LIN {X 0,Y 523.952,Z 221.716,A -85,B 0,C 180,E1 -4742.867,E2 -4742.867} C_VEL
LIN {X 0,Y 523.943,Z 221.723,A -85,B 0,C 180,E1 -4745.803,E2 -4745.803} C_VEL
LIN {X 0,Y 523.98,Z 221.883,A -85,B 0,C 180,E1 -4746.587,E2 -4746.587} C_VEL
LIN {X 0,Y 525.207,Z 229.637,A -85,B 0,C 180,E1 -4747.995,E2 -4747.995} C_VEL
LIN {X 0,Y 524.785,Z 247.797,A -85,B 0,C 180,E1 -4751.048,E2 -4751.048} C_VEL
LIN {X 0,Y 524.373,Z 265.937,A -85,B 0,C 180,E1 -4754.052,E2 -4754.052} C_VEL
LIN {X 0,Y 524.299,Z 270.906,A -85,B 0,C 180,E1 -4754.827,E2 -4754.827} C_VEL
LIN {X 0,Y 525.932,Z 281.44,A -85,B 0,C 180,E1 -4755.046,E2 -4755.046} C_VEL
LIN {X 0,Y 525.541,Z 378.256,A -85,B 0,C 180,E1 -4756.391,E2 -4756.391} C_VEL
LIN {X 0,Y 525.328,Z 391.632,A -85,B 0,C 180,E1 -4756.731,E2 -4756.731} C_VEL
LIN {X 0,Y 525.042,Z 404.968,A -85,B 0,C 180,E1 -4757.24,E2 -4757.24} C_VEL
LIN {X 0,Y 524.817,Z 416.488,A -85,B 0,C 180,E1 -4757.844,E2 -4757.844} C_VEL
LIN {X 0,Y 524.548,Z 427.759,A -85,B 0,C 180,E1 -4758.601,E2 -4758.601} C_VEL
LIN {X 0,Y 524.211,Z 438.203,A -85,B 0,C 180,E1 -4759.474,E2 -4759.474} C_VEL
LIN {X 0,Y 524.027,Z 446.741,A -85,B 0,C 180,E1 -4760.349,E2 -4760.349} C_VEL
LIN {X 0,Y 523.818,Z 454.616,A -85,B 0,C 180,E1 -4761.318,E2 -4761.318} C_VEL
LIN {X 0,Y 523.623,Z 462.304,A -85,B 0,C 180,E1 -4762.48,E2 -4762.48} C_VEL
LIN {X 0,Y 523.495,Z 469.387,A -85,B 0,C 180,E1 -4763.834,E2 -4763.834} C_VEL
LIN {X 0,Y 523.384,Z 474.097,A -85,B 0,C 180,E1 -4764.992,E2 -4764.992} C_VEL
LIN {X 0,Y 523.444,Z 477.697,A -85,B 0,C 180,E1 -4766.15,E2 -4766.15} C_VEL
LIN {X 0,Y 523.369,Z 479.553,A -85,B 0,C 180,E1 -4766.92,E2 -4766.92} C_VEL
LIN {X 0,Y 523.335,Z 480.944,A -85,B 0,C 180,E1 -4767.69,E2 -4767.69} C_VEL
LIN {X 0,Y 523.25,Z 482.542,A -85,B 0,C 180,E1 -4769.23,E2 -4769.23} C_VEL
LIN {X 0,Y 523.247,Z 482.758,A -85,B 0,C 180,E1 -4769.999,E2 -4769.999} C_VEL
LIN {X 0,Y 523.275,Z 481.938,A -85,B 0,C 180,E1 -4771.539,E2 -4771.539} C_VEL
LIN {X 0,Y 523.335,Z 480.947,A -85,B 0,C 180,E1 -4772.308,E2 -4772.308} C_VEL
LIN {X 0,Y 523.368,Z 479.556,A -85,B 0,C 180,E1 -4773.078,E2 -4773.078} C_VEL
LIN {X 0,Y 523.424,Z 476.63,A -85,B 0,C 180,E1 -4774.234,E2 -4774.234} C_VEL
LIN {X 0,Y 523.462,Z 472.667,A -85,B 0,C 180,E1 -4775.392,E2 -4775.392} C_VEL
LIN {X 0,Y 523.504,Z 466.596,A -85,B 0,C 180,E1 -4776.74,E2 -4776.74} C_VEL
LIN {X 0,Y 523.674,Z 459.907,A -85,B 0,C 180,E1 -4777.906,E2 -4777.906} C_VEL
LIN {X 0,Y 523.861,Z 451.635,A -85,B 0,C 180,E1 -4779.069,E2 -4779.069} C_VEL
LIN {X 0,Y 524.081,Z 443.153,A -85,B 0,C 180,E1 -4780.039,E2 -4780.039} C_VEL
LIN {X 0,Y 524.369,Z 432.668,A -85,B 0,C 180,E1 -4781.01,E2 -4781.01} C_VEL
LIN {X 0,Y 524.657,Z 422.414,A -85,B 0,C 180,E1 -4781.778,E2 -4781.778} C_VEL
LIN {X 0,Y 524.934,Z 410.912,A -85,B 0,C 180,E1 -4782.467,E2 -4782.467} C_VEL
LIN {X 0,Y 525.17,Z 399.214,A -85,B 0,C 180,E1 -4783.002,E2 -4783.002} C_VEL
LIN {X 0,Y 525.408,Z 386.643,A -85,B 0,C 180,E1 -4783.414,E2 -4783.414} C_VEL
LIN {X 0,Y 525.557,Z 373.865,A -85,B 0,C 180,E1 -4783.681,E2 -4783.681} C_VEL
LIN {X 0,Y 525.798,Z 280.337,A -85,B 0,C 180,E1 -4784.973,E2 -4784.973} C_VEL
LIN {X 0,Y 524.296,Z 270.856,A -85,B 0,C 180,E1 -4785.172,E2 -4785.172} C_VEL
LIN {X 0,Y 524.447,Z 259.751,A -85,B 0,C 180,E1 -4786.945,E2 -4786.945} C_VEL
LIN {X 0,Y 524.832,Z 242.691,A -85,B 0,C 180,E1 -4789.762,E2 -4789.762} C_VEL
LIN {X 0,Y 525.171,Z 229.26,A -85,B 0,C 180,E1 -4792.005,E2 -4792.005} C_VEL
LIN {X 0,Y 523.968,Z 221.828,A -85,B 0,C 180,E1 -4793.36,E2 -4793.36} C_VEL
LIN {X 0,Y 523.945,Z 221.72,A -85,B 0,C 180,E1 -4796.272,E2 -4796.272} C_VEL
LIN {X 0,Y 523.932,Z 221.718,A -85,B 0,C 180,E1 -4798.874,E2 -4798.874} C_VEL
LIN {X 0,Y 523.922,Z 221.723,A -85,B 0,C 180,E1 -4801.543,E2 -4801.543} C_VEL
LIN {X 0,Y 523.934,Z 221.722,A -85,B 0,C 180,E1 -4804.289,E2 -4804.289} C_VEL
LIN {X 0,Y 523.906,Z 221.718,A -85,B 0,C 180,E1 -4807.131,E2 -4807.131} C_VEL
LIN {X 0,Y 523.914,Z 221.724,A -85,B 0,C 180,E1 -4810.125,E2 -4810.125} C_VEL
LIN {X 0,Y 523.917,Z 221.723,A -85,B 0,C 180,E1 -4812.455,E2 -4812.455} C_VEL
LIN {X 0,Y 523.938,Z 221.715,A -85,B 0,C 180,E1 -4815.309,E2 -4815.309} C_VEL
LIN {X 0,Y 523.941,Z 221.72,A -85,B 0,C 180,E1 -4818.69,E2 -4818.69} C_VEL
LIN {X 0,Y 523.912,Z 221.719,A -85,B 0,C 180,E1 -4821.896,E2 -4821.896} C_VEL
LIN {X 0,Y 523.918,Z 221.722,A -85,B 0,C 180,E1 -4824.91,E2 -4824.91} C_VEL
LIN {X 0,Y 523.933,Z 221.716,A -85,B 0,C 180,E1 -4827.678,E2 -4827.678} C_VEL
LIN {X 0,Y 523.934,Z 221.725,A -85,B 0,C 180,E1 -4830.678,E2 -4830.678} C_VEL
LIN {X 0,Y 523.9,Z 221.72,A -85,B 0,C 180,E1 -4833.723,E2 -4833.723} C_VEL
LIN {X 0,Y 523.905,Z 221.72,A -85,B 0,C 180,E1 -4836.267,E2 -4836.267} C_VEL
LIN {X 0,Y 523.939,Z 221.721,A -85,B 0,C 180,E1 -4838.764,E2 -4838.764} C_VEL
LIN {X 0,Y 523.927,Z 221.721,A -85,B 0,C 180,E1 -4841.218,E2 -4841.218} C_VEL
LIN {X 0,Y 523.903,Z 221.722,A -85,B 0,C 180,E1 -4843.636,E2 -4843.636} C_VEL
LIN {X 0,Y 523.906,Z 221.717,A -85,B 0,C 180,E1 -4846.025,E2 -4846.025} C_VEL
LIN {X 0,Y 524.008,Z 221.706,A -85,B 0,C 180,E1 -4848.392,E2 -4848.392} C_VEL
LIN {X 0,Y 523.938,Z 221.721,A -85,B 0,C 180,E1 -4851.513,E2 -4851.513} C_VEL
LIN {X 0,Y 524.002,Z 221.711,A -85,B 0,C 180,E1 -4853.838,E2 -4853.838} C_VEL
LIN {X 0,Y 523.937,Z 221.723,A -85,B 0,C 180,E1 -4855.381,E2 -4855.381} C_VEL
LIN {X 0,Y 524.087,Z 221.704,A -85,B 0,C 180,E1 -4857.692,E2 -4857.692} C_VEL
LIN {X 0,Y 524.076,Z 221.7,A -85,B 0,C 180,E1 -4859.997,E2 -4859.997} C_VEL
LIN {X 0,Y 524.083,Z 221.698,A -85,B 0,C 180,E1 -4862.303,E2 -4862.303} C_VEL
LIN {X 0,Y 523.981,Z 221.713,A -85,B 0,C 180,E1 -4866.157,E2 -4866.157} C_VEL
LIN {X 0,Y 523.93,Z 221.718,A -85,B 0,C 180,E1 -4869.26,E2 -4869.26} C_VEL
LIN {X 0,Y 523.931,Z 221.719,A -85,B 0,C 180,E1 -4872.39,E2 -4872.39} C_VEL
LIN {X 0,Y 523.911,Z 221.723,A -85,B 0,C 180,E1 -4875.559,E2 -4875.559} C_VEL
LIN {X 0,Y 523.897,Z 221.727,A -85,B 0,C 180,E1 -4877.968,E2 -4877.968} C_VEL
LIN {X 0,Y 523.952,Z 221.719,A -85,B 0,C 180,E1 -4880.407,E2 -4880.407} C_VEL
LIN {X 0,Y 523.889,Z 221.722,A -85,B 0,C 180,E1 -4882.891,E2 -4882.891} C_VEL
LIN {X 0,Y 523.906,Z 221.719,A -85,B 0,C 180,E1 -4885.417,E2 -4885.417} C_VEL
LIN {X 0,Y 523.901,Z 221.725,A -85,B 0,C 180,E1 -4887.999,E2 -4887.999} C_VEL
LIN {X 0,Y 523.914,Z 221.722,A -85,B 0,C 180,E1 -4890.851,E2 -4890.851} C_VEL
LIN {X 0,Y 523.935,Z 221.717,A -85,B 0,C 180,E1 -4893.732,E2 -4893.732} C_VEL
LIN {X 0,Y 523.894,Z 221.728,A -85,B 0,C 180,E1 -4896.402,E2 -4896.402} C_VEL
LIN {X 0,Y 523.903,Z 221.725,A -85,B 0,C 180,E1 -4899.081,E2 -4899.081} C_VEL
LIN {X 0,Y 523.943,Z 221.719,A -85,B 0,C 180,E1 -4901.31,E2 -4901.31} C_VEL
LIN {X 0,Y 523.93,Z 221.726,A -85,B 0,C 180,E1 -4904.69,E2 -4904.69} C_VEL
LIN {X 0,Y 524.01,Z 221.942,A -85,B 0,C 180,E1 -4905.694,E2 -4905.694} C_VEL
LIN {X 0,Y 523.765,Z 225.215,A -85,B 0,C 180,E1 -4906.283,E2 -4906.283} C_VEL
LIN {X 0,Y 522.413,Z 228.497,A -85,B 0,C 180,E1 -4906.811,E2 -4906.811} C_VEL
LIN {X 0,Y 518.311,Z 236.117,A -85,B 0,C 180,E1 -4907.987,E2 -4907.987} C_VEL
LIN {X 0,Y 517.523,Z 239.242,A -85,B 0,C 180,E1 -4908.526,E2 -4908.526} C_VEL
LIN {X 0,Y 517.224,Z 256.986,A -85,B 0,C 180,E1 -4911.626,E2 -4911.626} C_VEL
LIN {X 0,Y 517.434,Z 258.712,A -85,B 0,C 180,E1 -4911.713,E2 -4911.713} C_VEL
LIN {X 0,Y 519.065,Z 267.751,A -85,B 0,C 180,E1 -4911.893,E2 -4911.893} C_VEL
LIN {X 0,Y 518.601,Z 364.846,A -85,B 0,C 180,E1 -4913.266,E2 -4913.266} C_VEL
LIN {X 0,Y 518.415,Z 377.895,A -85,B 0,C 180,E1 -4913.608,E2 -4913.608} C_VEL
LIN {X 0,Y 518.212,Z 390.252,A -85,B 0,C 180,E1 -4914.088,E2 -4914.088} C_VEL
LIN {X 0,Y 517.944,Z 401.526,A -85,B 0,C 180,E1 -4914.675,E2 -4914.675} C_VEL
LIN {X 0,Y 517.559,Z 412.829,A -85,B 0,C 180,E1 -4915.432,E2 -4915.432} C_VEL
LIN {X 0,Y 517.306,Z 422.833,A -85,B 0,C 180,E1 -4916.268,E2 -4916.268} C_VEL
LIN {X 0,Y 516.997,Z 432.757,A -85,B 0,C 180,E1 -4917.288,E2 -4917.288} C_VEL
LIN {X 0,Y 516.75,Z 441.634,A -85,B 0,C 180,E1 -4918.426,E2 -4918.426} C_VEL
LIN {X 0,Y 516.58,Z 448.883,A -85,B 0,C 180,E1 -4919.575,E2 -4919.575} C_VEL
LIN {X 0,Y 516.438,Z 454.473,A -85,B 0,C 180,E1 -4920.666,E2 -4920.666} C_VEL
LIN {X 0,Y 516.346,Z 459.559,A -85,B 0,C 180,E1 -4921.917,E2 -4921.917} C_VEL
LIN {X 0,Y 516.277,Z 463.773,A -85,B 0,C 180,E1 -4923.307,E2 -4923.307} C_VEL
LIN {X 0,Y 516.231,Z 465.648,A -85,B 0,C 180,E1 -4924.174,E2 -4924.174} C_VEL
LIN {X 0,Y 516.18,Z 467.035,A -85,B 0,C 180,E1 -4925.035,E2 -4925.035} C_VEL
LIN {X 0,Y 516.196,Z 467.919,A -85,B 0,C 180,E1 -4925.893,E2 -4925.893} C_VEL
LIN {X 0,Y 516.165,Z 468.305,A -85,B 0,C 180,E1 -4926.744,E2 -4926.744} C_VEL
LIN {X 0,Y 516.156,Z 468.166,A -85,B 0,C 180,E1 -4927.791,E2 -4927.791} C_VEL
LIN {X 0,Y 516.192,Z 466.722,A -85,B 0,C 180,E1 -4929.269,E2 -4929.269} C_VEL
LIN {X 0,Y 516.243,Z 465.293,A -85,B 0,C 180,E1 -4930.103,E2 -4930.103} C_VEL
LIN {X 0,Y 516.303,Z 462.244,A -85,B 0,C 180,E1 -4931.345,E2 -4931.345} C_VEL
LIN {X 0,Y 516.37,Z 458.075,A -85,B 0,C 180,E1 -4932.578,E2 -4932.578} C_VEL
LIN {X 0,Y 516.489,Z 451.624,A -85,B 0,C 180,E1 -4934.006,E2 -4934.006} C_VEL
LIN {X 0,Y 516.676,Z 444.589,A -85,B 0,C 180,E1 -4935.225,E2 -4935.225} C_VEL
LIN {X 0,Y 516.902,Z 437.397,A -85,B 0,C 180,E1 -4936.236,E2 -4936.236} C_VEL
LIN {X 0,Y 517.134,Z 428.727,A -85,B 0,C 180,E1 -4937.242,E2 -4937.242} C_VEL
LIN {X 0,Y 517.418,Z 418.012,A -85,B 0,C 180,E1 -4938.245,E2 -4938.245} C_VEL
LIN {X 0,Y 517.736,Z 407.363,A -85,B 0,C 180,E1 -4939.045,E2 -4939.045} C_VEL
LIN {X 0,Y 518.067,Z 395.552,A -85,B 0,C 180,E1 -4939.744,E2 -4939.744} C_VEL
LIN {X 0,Y 518.294,Z 383.305,A -85,B 0,C 180,E1 -4940.291,E2 -4940.291} C_VEL
LIN {X 0,Y 518.591,Z 370.453,A -85,B 0,C 180,E1 -4940.696,E2 -4940.696} C_VEL
LIN {X 0,Y 518.685,Z 357.828,A -85,B 0,C 180,E1 -4940.941,E2 -4940.941} C_VEL
LIN {X 0,Y 519.021,Z 267.402,A -85,B 0,C 180,E1 -4942.203,E2 -4942.203} C_VEL
LIN {X 0,Y 517.278,Z 257.789,A -85,B 0,C 180,E1 -4942.409,E2 -4942.409} C_VEL
LIN {X 0,Y 517.234,Z 256.652,A -85,B 0,C 180,E1 -4942.539,E2 -4942.539} C_VEL
LIN {X 0,Y 517.566,Z 244.544,A -85,B 0,C 180,E1 -4944.742,E2 -4944.742} C_VEL
LIN {X 0,Y 517.918,Z 228.732,A -85,B 0,C 180,E1 -4947.668,E2 -4947.668} C_VEL
LIN {X 0,Y 516.991,Z 222.635,A -85,B 0,C 180,E1 -4948.905,E2 -4948.905} C_VEL
LIN {X 0,Y 517.058,Z 222.578,A -85,B 0,C 180,E1 -4950.779,E2 -4950.779} C_VEL
LIN {X 0,Y 516.981,Z 222.589,A -85,B 0,C 180,E1 -4953.118,E2 -4953.118} C_VEL
LIN {X 0,Y 516.966,Z 222.585,A -85,B 0,C 180,E1 -4956.244,E2 -4956.244} C_VEL
LIN {X 0,Y 516.915,Z 222.597,A -85,B 0,C 180,E1 -4959.391,E2 -4959.391} C_VEL
LIN {X 0,Y 516.946,Z 222.591,A -85,B 0,C 180,E1 -4961.826,E2 -4961.826} C_VEL
LIN {X 0,Y 516.906,Z 222.593,A -85,B 0,C 180,E1 -4965.147,E2 -4965.147} C_VEL
LIN {X 0,Y 516.889,Z 222.598,A -85,B 0,C 180,E1 -4968.224,E2 -4968.224} C_VEL
LIN {X 0,Y 516.876,Z 222.595,A -85,B 0,C 180,E1 -4970.703,E2 -4970.703} C_VEL
LIN {X 0,Y 516.856,Z 222.604,A -85,B 0,C 180,E1 -4974.075,E2 -4974.075} C_VEL
LIN {X 0,Y 516.863,Z 222.599,A -85,B 0,C 180,E1 -4976.662,E2 -4976.662} C_VEL
LIN {X 0,Y 516.878,Z 222.591,A -85,B 0,C 180,E1 -4979.526,E2 -4979.526} C_VEL
LIN {X 0,Y 516.863,Z 222.602,A -85,B 0,C 180,E1 -4982.546,E2 -4982.546} C_VEL
LIN {X 0,Y 516.826,Z 222.596,A -85,B 0,C 180,E1 -4985.331,E2 -4985.331} C_VEL
LIN {X 0,Y 516.844,Z 222.606,A -85,B 0,C 180,E1 -4988.72,E2 -4988.72} C_VEL
LIN {X 0,Y 516.826,Z 222.598,A -85,B 0,C 180,E1 -4991.784,E2 -4991.784} C_VEL
LIN {X 0,Y 516.871,Z 222.601,A -85,B 0,C 180,E1 -4995.01,E2 -4995.01} C_VEL
LIN {X 0,Y 516.832,Z 222.603,A -85,B 0,C 180,E1 -4998.409,E2 -4998.409} C_VEL
LIN {X 0,Y 516.855,Z 222.595,A -85,B 0,C 180,E1 -5001.287,E2 -5001.287} C_VEL
LIN {X 0,Y 516.85,Z 222.597,A -85,B 0,C 180,E1 -5004.223,E2 -5004.223} C_VEL
LIN {X 0,Y 516.863,Z 222.605,A -85,B 0,C 180,E1 -5007.055,E2 -5007.055} C_VEL
LIN {X 0,Y 516.838,Z 222.595,A -85,B 0,C 180,E1 -5009.797,E2 -5009.797} C_VEL
LIN {X 0,Y 516.855,Z 222.59,A -85,B 0,C 180,E1 -5012.467,E2 -5012.467} C_VEL
LIN {X 0,Y 516.859,Z 222.603,A -85,B 0,C 180,E1 -5015.649,E2 -5015.649} C_VEL
LIN {X 0,Y 516.875,Z 222.594,A -85,B 0,C 180,E1 -5018.465,E2 -5018.465} C_VEL
LIN {X 0,Y 516.881,Z 222.59,A -85,B 0,C 180,E1 -5020.958,E2 -5020.958} C_VEL
LIN {X 0,Y 516.875,Z 222.589,A -85,B 0,C 180,E1 -5023.412,E2 -5023.412} C_VEL
LIN {X 0,Y 516.876,Z 222.602,A -85,B 0,C 180,E1 -5025.836,E2 -5025.836} C_VEL
LIN {X 0,Y 516.922,Z 222.592,A -85,B 0,C 180,E1 -5028.236,E2 -5028.236} C_VEL
LIN {X 0,Y 516.926,Z 222.588,A -85,B 0,C 180,E1 -5031.402,E2 -5031.402} C_VEL
LIN {X 0,Y 516.983,Z 222.575,A -85,B 0,C 180,E1 -5034.542,E2 -5034.542} C_VEL
LIN {X 0,Y 517.071,Z 222.571,A -85,B 0,C 180,E1 -5037.666,E2 -5037.666} C_VEL
LIN {X 0,Y 517.068,Z 222.572,A -85,B 0,C 180,E1 -5040.781,E2 -5040.781} C_VEL
LIN {X 0,Y 516.946,Z 222.581,A -85,B 0,C 180,E1 -5043.12,E2 -5043.12} C_VEL
LIN {X 0,Y 516.986,Z 222.579,A -85,B 0,C 180,E1 -5046.246,E2 -5046.246} C_VEL
LIN {X 0,Y 516.92,Z 222.589,A -85,B 0,C 180,E1 -5049.392,E2 -5049.392} C_VEL
LIN {X 0,Y 516.959,Z 222.585,A -85,B 0,C 180,E1 -5051.809,E2 -5051.809} C_VEL
LIN {X 0,Y 516.943,Z 222.582,A -85,B 0,C 180,E1 -5055.145,E2 -5055.145} C_VEL
LIN {X 0,Y 516.919,Z 222.59,A -85,B 0,C 180,E1 -5058.225,E2 -5058.225} C_VEL
LIN {X 0,Y 516.911,Z 222.598,A -85,B 0,C 180,E1 -5060.704,E2 -5060.704} C_VEL
LIN {X 0,Y 516.893,Z 222.586,A -85,B 0,C 180,E1 -5064.075,E2 -5064.075} C_VEL
LIN {X 0,Y 516.902,Z 222.594,A -85,B 0,C 180,E1 -5066.661,E2 -5066.661} C_VEL
LIN {X 0,Y 516.894,Z 222.594,A -85,B 0,C 180,E1 -5069.52,E2 -5069.52} C_VEL
LIN {X 0,Y 516.902,Z 222.59,A -85,B 0,C 180,E1 -5072.544,E2 -5072.544} C_VEL
LIN {X 0,Y 516.869,Z 222.605,A -85,B 0,C 180,E1 -5075.329,E2 -5075.329} C_VEL
LIN {X 0,Y 516.886,Z 222.594,A -85,B 0,C 180,E1 -5077.943,E2 -5077.943} C_VEL
LIN {X 0,Y 516.873,Z 222.596,A -85,B 0,C 180,E1 -5080.744,E2 -5080.744} C_VEL
LIN {X 0,Y 516.89,Z 222.599,A -85,B 0,C 180,E1 -5083.904,E2 -5083.904} C_VEL
LIN {X 0,Y 516.89,Z 222.595,A -85,B 0,C 180,E1 -5086.108,E2 -5086.108} C_VEL
LIN {X 0,Y 516.862,Z 222.599,A -85,B 0,C 180,E1 -5089.256,E2 -5089.256} C_VEL
LIN {X 0,Y 516.869,Z 222.6,A -85,B 0,C 180,E1 -5092.274,E2 -5092.274} C_VEL
LIN {X 0,Y 516.889,Z 222.595,A -85,B 0,C 180,E1 -5095.175,E2 -5095.175} C_VEL
LIN {X 0,Y 516.882,Z 222.603,A -85,B 0,C 180,E1 -5097.975,E2 -5097.975} C_VEL
LIN {X 0,Y 516.928,Z 222.592,A -85,B 0,C 180,E1 -5100.695,E2 -5100.695} C_VEL
LIN {X 0,Y 516.91,Z 222.595,A -85,B 0,C 180,E1 -5103.814,E2 -5103.814} C_VEL
LIN {X 0,Y 516.94,Z 222.731,A -85,B 0,C 180,E1 -5106.408,E2 -5106.408} C_VEL
LIN {X 0,Y 518.257,Z 230.758,A -85,B 0,C 180,E1 -5107.894,E2 -5107.894} C_VEL
LIN {X 0,Y 517.843,Z 245.281,A -85,B 0,C 180,E1 -5110.372,E2 -5110.372} C_VEL
LIN {X 0,Y 517.469,Z 261.007,A -85,B 0,C 180,E1 -5113.022,E2 -5113.022} C_VEL
LIN {X 0,Y 517.277,Z 270.787,A -85,B 0,C 180,E1 -5114.614,E2 -5114.614} C_VEL
LIN {X 0,Y 519.075,Z 282.522,A -85,B 0,C 180,E1 -5114.861,E2 -5114.861} C_VEL
LIN {X 0,Y 518.665,Z 378.097,A -85,B 0,C 180,E1 -5116.207,E2 -5116.207} C_VEL
LIN {X 0,Y 518.424,Z 391.496,A -85,B 0,C 180,E1 -5116.551,E2 -5116.551} C_VEL
LIN {X 0,Y 518.128,Z 404.842,A -85,B 0,C 180,E1 -5117.067,E2 -5117.067} C_VEL
LIN {X 0,Y 517.878,Z 416.092,A -85,B 0,C 180,E1 -5117.662,E2 -5117.662} C_VEL
LIN {X 0,Y 517.568,Z 427.645,A -85,B 0,C 180,E1 -5118.446,E2 -5118.446} C_VEL
LIN {X 0,Y 517.206,Z 438.092,A -85,B 0,C 180,E1 -5119.33,E2 -5119.33} C_VEL
LIN {X 0,Y 516.98,Z 446.633,A -85,B 0,C 180,E1 -5120.216,E2 -5120.216} C_VEL
LIN {X 0,Y 516.756,Z 454.51,A -85,B 0,C 180,E1 -5121.198,E2 -5121.198} C_VEL
LIN {X 0,Y 516.551,Z 462.2,A -85,B 0,C 180,E1 -5122.376,E2 -5122.376} C_VEL
LIN {X 0,Y 516.405,Z 469.285,A -85,B 0,C 180,E1 -5123.749,E2 -5123.749} C_VEL
LIN {X 0,Y 516.314,Z 473.997,A -85,B 0,C 180,E1 -5124.923,E2 -5124.923} C_VEL
LIN {X 0,Y 516.353,Z 477.598,A -85,B 0,C 180,E1 -5126.097,E2 -5126.097} C_VEL
LIN {X 0,Y 516.284,Z 479.454,A -85,B 0,C 180,E1 -5126.878,E2 -5126.878} C_VEL
LIN {X 0,Y 516.262,Z 480.846,A -85,B 0,C 180,E1 -5127.659,E2 -5127.659} C_VEL
LIN {X 0,Y 516.16,Z 482.444,A -85,B 0,C 180,E1 -5129.219,E2 -5129.219} C_VEL
LIN {X 0,Y 516.155,Z 482.66,A -85,B 0,C 180,E1 -5129.999,E2 -5129.999} C_VEL
LIN {X 0,Y 516.192,Z 481.839,A -85,B 0,C 180,E1 -5131.56,E2 -5131.56} C_VEL
LIN {X 0,Y 516.261,Z 480.847,A -85,B 0,C 180,E1 -5132.34,E2 -5132.34} C_VEL
LIN {X 0,Y 516.283,Z 479.456,A -85,B 0,C 180,E1 -5133.121,E2 -5133.121} C_VEL
LIN {X 0,Y 516.313,Z 476.528,A -85,B 0,C 180,E1 -5134.293,E2 -5134.293} C_VEL
LIN {X 0,Y 516.398,Z 472.564,A -85,B 0,C 180,E1 -5135.466,E2 -5135.466} C_VEL
LIN {X 0,Y 516.423,Z 467.358,A -85,B 0,C 180,E1 -5136.663,E2 -5136.663} C_VEL
LIN {X 0,Y 516.583,Z 461.034,A -85,B 0,C 180,E1 -5137.818,E2 -5137.818} C_VEL
LIN {X 0,Y 516.772,Z 453.014,A -85,B 0,C 180,E1 -5138.997,E2 -5138.997} C_VEL
LIN {X 0,Y 517.026,Z 444.839,A -85,B 0,C 180,E1 -5139.98,E2 -5139.98} C_VEL
LIN {X 0,Y 517.336,Z 434.868,A -85,B 0,C 180,E1 -5140.963,E2 -5140.963} C_VEL
LIN {X 0,Y 517.646,Z 425.024,A -85,B 0,C 180,E1 -5141.75,E2 -5141.75} C_VEL
LIN {X 0,Y 517.914,Z 413.875,A -85,B 0,C 180,E1 -5142.465,E2 -5142.465} C_VEL
LIN {X 0,Y 518.197,Z 401.437,A -85,B 0,C 180,E1 -5143.08,E2 -5143.08} C_VEL
LIN {X 0,Y 518.502,Z 389.187,A -85,B 0,C 180,E1 -5143.521,E2 -5143.521} C_VEL
LIN {X 0,Y 518.639,Z 376.686,A -85,B 0,C 180,E1 -5143.817,E2 -5143.817} C_VEL
LIN {X 0,Y 519.048,Z 281.84,A -85,B 0,C 180,E1 -5145.149,E2 -5145.149} C_VEL
LIN {X 0,Y 517.261,Z 270.774,A -85,B 0,C 180,E1 -5145.381,E2 -5145.381} C_VEL
LIN {X 0,Y 517.493,Z 259.643,A -85,B 0,C 180,E1 -5147.18,E2 -5147.18} C_VEL
LIN {X 0,Y 517.973,Z 240.109,A -85,B 0,C 180,E1 -5150.452,E2 -5150.452} C_VEL
LIN {X 0,Y 518.205,Z 230.362,A -85,B 0,C 180,E1 -5152.107,E2 -5152.107} C_VEL
LIN {X 0,Y 516.931,Z 222.671,A -85,B 0,C 180,E1 -5153.538,E2 -5153.538} C_VEL
LIN {X 0,Y 516.913,Z 222.594,A -85,B 0,C 180,E1 -5156.657,E2 -5156.657} C_VEL
LIN {X 0,Y 516.912,Z 222.598,A -85,B 0,C 180,E1 -5159.522,E2 -5159.522} C_VEL
LIN {X 0,Y 516.899,Z 222.595,A -85,B 0,C 180,E1 -5162.542,E2 -5162.542} C_VEL
LIN {X 0,Y 516.866,Z 222.599,A -85,B 0,C 180,E1 -5165.328,E2 -5165.328} C_VEL
LIN {X 0,Y 516.88,Z 222.601,A -85,B 0,C 180,E1 -5167.941,E2 -5167.941} C_VEL
LIN {X 0,Y 516.865,Z 222.598,A -85,B 0,C 180,E1 -5170.742,E2 -5170.742} C_VEL
LIN {X 0,Y 516.856,Z 222.599,A -85,B 0,C 180,E1 -5172.833,E2 -5172.833} C_VEL
LIN {X 0,Y 516.897,Z 222.593,A -85,B 0,C 180,E1 -5175.005,E2 -5175.005} C_VEL
LIN {X 0,Y 516.904,Z 222.599,A -85,B 0,C 180,E1 -5178.399,E2 -5178.399} C_VEL
LIN {X 0,Y 516.876,Z 222.594,A -85,B 0,C 180,E1 -5181.282,E2 -5181.282} C_VEL
LIN {X 0,Y 516.866,Z 222.601,A -85,B 0,C 180,E1 -5184.217,E2 -5184.217} C_VEL
LIN {X 0,Y 516.88,Z 222.598,A -85,B 0,C 180,E1 -5187.05,E2 -5187.05} C_VEL
LIN {X 0,Y 516.865,Z 222.596,A -85,B 0,C 180,E1 -5189.793,E2 -5189.793} C_VEL
LIN {X 0,Y 516.873,Z 222.6,A -85,B 0,C 180,E1 -5192.462,E2 -5192.462} C_VEL
LIN {X 0,Y 516.844,Z 222.605,A -85,B 0,C 180,E1 -5195.066,E2 -5195.066} C_VEL
LIN {X 0,Y 516.867,Z 222.596,A -85,B 0,C 180,E1 -5197.619,E2 -5197.619} C_VEL
LIN {X 0,Y 516.916,Z 222.59,A -85,B 0,C 180,E1 -5200.127,E2 -5200.127} C_VEL
LIN {X 0,Y 516.889,Z 222.593,A -85,B 0,C 180,E1 -5202.593,E2 -5202.593} C_VEL
LIN {X 0,Y 516.926,Z 222.597,A -85,B 0,C 180,E1 -5205.027,E2 -5205.027} C_VEL
LIN {X 0,Y 516.961,Z 222.584,A -85,B 0,C 180,E1 -5208.231,E2 -5208.231} C_VEL
LIN {X 0,Y 516.912,Z 222.596,A -85,B 0,C 180,E1 -5211.396,E2 -5211.396} C_VEL
LIN {X 0,Y 516.972,Z 222.587,A -85,B 0,C 180,E1 -5213.754,E2 -5213.754} C_VEL
LIN {X 0,Y 516.931,Z 222.586,A -85,B 0,C 180,E1 -5216.88,E2 -5216.88} C_VEL
LIN {X 0,Y 517.078,Z 222.575,A -85,B 0,C 180,E1 -5219.219,E2 -5219.219} C_VEL
LIN {X 0,Y 517.053,Z 222.574,A -85,B 0,C 180,E1 -5222.334,E2 -5222.334} C_VEL
LIN {X 0,Y 516.962,Z 222.589,A -85,B 0,C 180,E1 -5225.458,E2 -5225.458} C_VEL
LIN {X 0,Y 516.905,Z 222.591,A -85,B 0,C 180,E1 -5228.598,E2 -5228.598} C_VEL
LIN {X 0,Y 516.917,Z 222.598,A -85,B 0,C 180,E1 -5231.793,E2 -5231.793} C_VEL
LIN {X 0,Y 516.922,Z 222.59,A -85,B 0,C 180,E1 -5235.141,E2 -5235.141} C_VEL
LIN {X 0,Y 516.859,Z 222.605,A -85,B 0,C 180,E1 -5238.221,E2 -5238.221} C_VEL
LIN {X 0,Y 516.893,Z 222.595,A -85,B 0,C 180,E1 -5240.699,E2 -5240.699} C_VEL
LIN {X 0,Y 516.868,Z 222.603,A -85,B 0,C 180,E1 -5244.07,E2 -5244.07} C_VEL
LIN {X 0,Y 516.875,Z 222.6,A -85,B 0,C 180,E1 -5246.657,E2 -5246.657} C_VEL
LIN {X 0,Y 516.885,Z 222.593,A -85,B 0,C 180,E1 -5249.521,E2 -5249.521} C_VEL
LIN {X 0,Y 516.87,Z 222.603,A -85,B 0,C 180,E1 -5252.541,E2 -5252.541} C_VEL
LIN {X 0,Y 516.855,Z 222.599,A -85,B 0,C 180,E1 -5255.33,E2 -5255.33} C_VEL
LIN {X 0,Y 516.854,Z 222.599,A -85,B 0,C 180,E1 -5257.941,E2 -5257.941} C_VEL
LIN {X 0,Y 516.875,Z 222.604,A -85,B 0,C 180,E1 -5260.737,E2 -5260.737} C_VEL
LIN {X 0,Y 516.853,Z 222.603,A -85,B 0,C 180,E1 -5263.901,E2 -5263.901} C_VEL
LIN {X 0,Y 516.942,Z 222.726,A -85,B 0,C 180,E1 -5265.535,E2 -5265.535} C_VEL
LIN {X 0,Y 517.7,Z 227.862,A -85,B 0,C 180,E1 -5266.514,E2 -5266.514} C_VEL
LIN {X 0,Y 517.523,Z 239.242,A -85,B 0,C 180,E1 -5268.526,E2 -5268.526} C_VEL
LIN {X 0,Y 516.78,Z 242.514,A -85,B 0,C 180,E1 -5269.073,E2 -5269.073} C_VEL
LIN {X 0,Y 511.465,Z 252.389,A -85,B 0,C 180,E1 -5270.641,E2 -5270.641} C_VEL
LIN {X 0,Y 510.373,Z 255.577,A -85,B 0,C 180,E1 -5271.173,E2 -5271.173} C_VEL
LIN {X 0,Y 510.255,Z 256.657,A -85,B 0,C 180,E1 -5271.35,E2 -5271.35} C_VEL
LIN {X 0,Y 510.286,Z 257.654,A -85,B 0,C 180,E1 -5271.463,E2 -5271.463} C_VEL
LIN {X 0,Y 512.22,Z 268.774,A -85,B 0,C 180,E1 -5271.699,E2 -5271.699} C_VEL
LIN {X 0,Y 511.718,Z 365.201,A -85,B 0,C 180,E1 -5273.084,E2 -5273.084} C_VEL
LIN {X 0,Y 511.501,Z 378.295,A -85,B 0,C 180,E1 -5273.435,E2 -5273.435} C_VEL
LIN {X 0,Y 511.305,Z 390.217,A -85,B 0,C 180,E1 -5273.905,E2 -5273.905} C_VEL
LIN {X 0,Y 510.996,Z 402.179,A -85,B 0,C 180,E1 -5274.54,E2 -5274.54} C_VEL
LIN {X 0,Y 510.601,Z 413.104,A -85,B 0,C 180,E1 -5275.286,E2 -5275.286} C_VEL
LIN {X 0,Y 510.299,Z 423.97,A -85,B 0,C 180,E1 -5276.218,E2 -5276.218} C_VEL
LIN {X 0,Y 509.971,Z 433.267,A -85,B 0,C 180,E1 -5277.201,E2 -5277.201} C_VEL
LIN {X 0,Y 509.697,Z 442.379,A -85,B 0,C 180,E1 -5278.402,E2 -5278.402} C_VEL
LIN {X 0,Y 509.509,Z 449.376,A -85,B 0,C 180,E1 -5279.542,E2 -5279.542} C_VEL
LIN {X 0,Y 509.343,Z 455.299,A -85,B 0,C 180,E1 -5280.738,E2 -5280.738} C_VEL
LIN {X 0,Y 509.254,Z 460.298,A -85,B 0,C 180,E1 -5282.026,E2 -5282.026} C_VEL
LIN {X 0,Y 509.192,Z 464.089,A -85,B 0,C 180,E1 -5283.349,E2 -5283.349} C_VEL
LIN {X 0,Y 509.091,Z 466.647,A -85,B 0,C 180,E1 -5284.663,E2 -5284.663} C_VEL
LIN {X 0,Y 509.096,Z 467.832,A -85,B 0,C 180,E1 -5285.65,E2 -5285.65} C_VEL
LIN {X 0,Y 509.075,Z 468.328,A -85,B 0,C 180,E1 -5286.4,E2 -5286.4} C_VEL
LIN {X 0,Y 509.071,Z 468.34,A -85,B 0,C 180,E1 -5287.652,E2 -5287.652} C_VEL
LIN {X 0,Y 509.075,Z 467.289,A -85,B 0,C 180,E1 -5288.966,E2 -5288.966} C_VEL
LIN {X 0,Y 509.138,Z 465.998,A -85,B 0,C 180,E1 -5289.813,E2 -5289.813} C_VEL
LIN {X 0,Y 509.208,Z 463.223,A -85,B 0,C 180,E1 -5291.075,E2 -5291.075} C_VEL
LIN {X 0,Y 509.265,Z 459.354,A -85,B 0,C 180,E1 -5292.327,E2 -5292.327} C_VEL
LIN {X 0,Y 509.377,Z 454.291,A -85,B 0,C 180,E1 -5293.571,E2 -5293.571} C_VEL
LIN {X 0,Y 509.557,Z 447.491,A -85,B 0,C 180,E1 -5294.881,E2 -5294.881} C_VEL
LIN {X 0,Y 509.799,Z 439.894,A -85,B 0,C 180,E1 -5296.04,E2 -5296.04} C_VEL
LIN {X 0,Y 510.04,Z 431.713,A -85,B 0,C 180,E1 -5297.062,E2 -5297.062} C_VEL
LIN {X 0,Y 510.332,Z 421.743,A -85,B 0,C 180,E1 -5298.079,E2 -5298.079} C_VEL
LIN {X 0,Y 510.645,Z 411.942,A -85,B 0,C 180,E1 -5298.891,E2 -5298.891} C_VEL
LIN {X 0,Y 511.007,Z 401.324,A -85,B 0,C 180,E1 -5299.601,E2 -5299.601} C_VEL
LIN {X 0,Y 511.28,Z 389.722,A -85,B 0,C 180,E1 -5300.207,E2 -5300.207} C_VEL
LIN {X 0,Y 511.539,Z 376.813,A -85,B 0,C 180,E1 -5300.703,E2 -5300.703} C_VEL
LIN {X 0,Y 511.722,Z 364.511,A -85,B 0,C 180,E1 -5301.02,E2 -5301.02} C_VEL
LIN {X 0,Y 512.069,Z 267.751,A -85,B 0,C 180,E1 -5302.41,E2 -5302.41} C_VEL
LIN {X 0,Y 510.277,Z 257.584,A -85,B 0,C 180,E1 -5302.64,E2 -5302.64} C_VEL
LIN {X 0,Y 510.567,Z 246.346,A -85,B 0,C 180,E1 -5304.669,E2 -5304.669} C_VEL
LIN {X 0,Y 510.985,Z 230.504,A -85,B 0,C 180,E1 -5307.636,E2 -5307.636} C_VEL
LIN {X 0,Y 510.001,Z 223.506,A -85,B 0,C 180,E1 -5309.063,E2 -5309.063} C_VEL
LIN {X 0,Y 510.029,Z 223.454,A -85,B 0,C 180,E1 -5310.79,E2 -5310.79} C_VEL
LIN {X 0,Y 509.924,Z 223.468,A -85,B 0,C 180,E1 -5313.161,E2 -5313.161} C_VEL
LIN {X 0,Y 509.917,Z 223.463,A -85,B 0,C 180,E1 -5316.331,E2 -5316.331} C_VEL
LIN {X 0,Y 509.877,Z 223.468,A -85,B 0,C 180,E1 -5318.721,E2 -5318.721} C_VEL
LIN {X 0,Y 509.914,Z 223.465,A -85,B 0,C 180,E1 -5321.932,E2 -5321.932} C_VEL
LIN {X 0,Y 509.857,Z 223.472,A -85,B 0,C 180,E1 -5325.243,E2 -5325.243} C_VEL
LIN {X 0,Y 509.852,Z 223.478,A -85,B 0,C 180,E1 -5328.003,E2 -5328.003} C_VEL
LIN {X 0,Y 509.814,Z 223.474,A -85,B 0,C 180,E1 -5331.004,E2 -5331.004} C_VEL
LIN {X 0,Y 509.787,Z 223.48,A -85,B 0,C 180,E1 -5333.566,E2 -5333.566} C_VEL
LIN {X 0,Y 509.85,Z 223.476,A -85,B 0,C 180,E1 -5336.374,E2 -5336.374} C_VEL
LIN {X 0,Y 509.826,Z 223.472,A -85,B 0,C 180,E1 -5339.754,E2 -5339.754} C_VEL
LIN {X 0,Y 509.815,Z 223.477,A -85,B 0,C 180,E1 -5342.772,E2 -5342.772} C_VEL
LIN {X 0,Y 509.784,Z 223.473,A -85,B 0,C 180,E1 -5345.579,E2 -5345.579} C_VEL
LIN {X 0,Y 509.787,Z 223.485,A -85,B 0,C 180,E1 -5348.344,E2 -5348.344} C_VEL
LIN {X 0,Y 509.781,Z 223.475,A -85,B 0,C 180,E1 -5351.433,E2 -5351.433} C_VEL
LIN {X 0,Y 509.815,Z 223.48,A -85,B 0,C 180,E1 -5354.673,E2 -5354.673} C_VEL
LIN {X 0,Y 509.768,Z 223.481,A -85,B 0,C 180,E1 -5357.509,E2 -5357.509} C_VEL
LIN {X 0,Y 509.811,Z 223.476,A -85,B 0,C 180,E1 -5360.649,E2 -5360.649} C_VEL
LIN {X 0,Y 509.804,Z 223.475,A -85,B 0,C 180,E1 -5363.65,E2 -5363.65} C_VEL
LIN {X 0,Y 509.824,Z 223.475,A -85,B 0,C 180,E1 -5366.541,E2 -5366.541} C_VEL
LIN {X 0,Y 509.808,Z 223.476,A -85,B 0,C 180,E1 -5369.336,E2 -5369.336} C_VEL
LIN {X 0,Y 509.814,Z 223.467,A -85,B 0,C 180,E1 -5372.054,E2 -5372.054} C_VEL
LIN {X 0,Y 509.782,Z 223.477,A -85,B 0,C 180,E1 -5374.703,E2 -5374.703} C_VEL
LIN {X 0,Y 509.815,Z 223.483,A -85,B 0,C 180,E1 -5377.462,E2 -5377.462} C_VEL
LIN {X 0,Y 509.908,Z 223.462,A -85,B 0,C 180,E1 -5379.848,E2 -5379.848} C_VEL
LIN {X 0,Y 509.844,Z 223.461,A -85,B 0,C 180,E1 -5383.177,E2 -5383.177} C_VEL
LIN {X 0,Y 509.847,Z 223.474,A -85,B 0,C 180,E1 -5385.637,E2 -5385.637} C_VEL
LIN {X 0,Y 509.885,Z 223.47,A -85,B 0,C 180,E1 -5388.134,E2 -5388.134} C_VEL
LIN {X 0,Y 509.88,Z 223.465,A -85,B 0,C 180,E1 -5391.282,E2 -5391.282} C_VEL
LIN {X 0,Y 509.92,Z 223.458,A -85,B 0,C 180,E1 -5393.673,E2 -5393.673} C_VEL
LIN {X 0,Y 509.889,Z 223.463,A -85,B 0,C 180,E1 -5396.842,E2 -5396.842} C_VEL
LIN {X 0,Y 509.928,Z 223.465,A -85,B 0,C 180,E1 -5398.423,E2 -5398.423} C_VEL
LIN {X 0,Y 510.02,Z 223.449,A -85,B 0,C 180,E1 -5400.792,E2 -5400.792} C_VEL
LIN {X 0,Y 510.041,Z 223.449,A -85,B 0,C 180,E1 -5402.372,E2 -5402.372} C_VEL
LIN {X 0,Y 509.94,Z 223.457,A -85,B 0,C 180,E1 -5406.333,E2 -5406.333} C_VEL
LIN {X 0,Y 509.882,Z 223.472,A -85,B 0,C 180,E1 -5408.723,E2 -5408.723} C_VEL
LIN {X 0,Y 509.911,Z 223.464,A -85,B 0,C 180,E1 -5411.934,E2 -5411.934} C_VEL
LIN {X 0,Y 509.902,Z 223.458,A -85,B 0,C 180,E1 -5415.244,E2 -5415.244} C_VEL
LIN {X 0,Y 509.864,Z 223.472,A -85,B 0,C 180,E1 -5418.486,E2 -5418.486} C_VEL
LIN {X 0,Y 509.853,Z 223.476,A -85,B 0,C 180,E1 -5421.004,E2 -5421.004} C_VEL
LIN {X 0,Y 509.826,Z 223.467,A -85,B 0,C 180,E1 -5423.566,E2 -5423.566} C_VEL
LIN {X 0,Y 509.883,Z 223.465,A -85,B 0,C 180,E1 -5426.371,E2 -5426.371} C_VEL
LIN {X 0,Y 509.86,Z 223.468,A -85,B 0,C 180,E1 -5429.753,E2 -5429.753} C_VEL
LIN {X 0,Y 509.854,Z 223.47,A -85,B 0,C 180,E1 -5432.77,E2 -5432.77} C_VEL
LIN {X 0,Y 509.829,Z 223.477,A -85,B 0,C 180,E1 -5435.578,E2 -5435.578} C_VEL
LIN {X 0,Y 509.857,Z 223.468,A -85,B 0,C 180,E1 -5438.339,E2 -5438.339} C_VEL
LIN {X 0,Y 509.85,Z 223.479,A -85,B 0,C 180,E1 -5441.428,E2 -5441.428} C_VEL
LIN {X 0,Y 509.849,Z 223.471,A -85,B 0,C 180,E1 -5444.671,E2 -5444.671} C_VEL
LIN {X 0,Y 509.811,Z 223.48,A -85,B 0,C 180,E1 -5447.507,E2 -5447.507} C_VEL
LIN {X 0,Y 509.841,Z 223.472,A -85,B 0,C 180,E1 -5450.647,E2 -5450.647} C_VEL
LIN {X 0,Y 509.818,Z 223.481,A -85,B 0,C 180,E1 -5453.646,E2 -5453.646} C_VEL
LIN {X 0,Y 509.867,Z 223.47,A -85,B 0,C 180,E1 -5456.539,E2 -5456.539} C_VEL
LIN {X 0,Y 509.849,Z 223.471,A -85,B 0,C 180,E1 -5459.334,E2 -5459.334} C_VEL
LIN {X 0,Y 509.892,Z 223.472,A -85,B 0,C 180,E1 -5462.054,E2 -5462.054} C_VEL
LIN {X 0,Y 509.821,Z 223.48,A -85,B 0,C 180,E1 -5464.7,E2 -5464.7} C_VEL
LIN {X 0,Y 509.872,Z 223.582,A -85,B 0,C 180,E1 -5466.223,E2 -5466.223} C_VEL
LIN {X 0,Y 511.287,Z 231.878,A -85,B 0,C 180,E1 -5467.789,E2 -5467.789} C_VEL
LIN {X 0,Y 511.023,Z 242.12,A -85,B 0,C 180,E1 -5469.567,E2 -5469.567} C_VEL
LIN {X 0,Y 510.525,Z 259.705,A -85,B 0,C 180,E1 -5472.577,E2 -5472.577} C_VEL
LIN {X 0,Y 510.281,Z 270.685,A -85,B 0,C 180,E1 -5474.398,E2 -5474.398} C_VEL
LIN {X 0,Y 512.223,Z 283.007,A -85,B 0,C 180,E1 -5474.662,E2 -5474.662} C_VEL
LIN {X 0,Y 511.771,Z 379.1,A -85,B 0,C 180,E1 -5476.043,E2 -5476.043} C_VEL
LIN {X 0,Y 511.497,Z 392.121,A -85,B 0,C 180,E1 -5476.39,E2 -5476.39} C_VEL
LIN {X 0,Y 511.195,Z 404.716,A -85,B 0,C 180,E1 -5476.888,E2 -5476.888} C_VEL
LIN {X 0,Y 510.918,Z 416.09,A -85,B 0,C 180,E1 -5477.498,E2 -5477.498} C_VEL
LIN {X 0,Y 510.602,Z 427.531,A -85,B 0,C 180,E1 -5478.286,E2 -5478.286} C_VEL
LIN {X 0,Y 510.217,Z 437.982,A -85,B 0,C 180,E1 -5479.182,E2 -5479.182} C_VEL
LIN {X 0,Y 509.954,Z 446.525,A -85,B 0,C 180,E1 -5480.08,E2 -5480.08} C_VEL
LIN {X 0,Y 509.69,Z 454.404,A -85,B 0,C 180,E1 -5481.075,E2 -5481.075} C_VEL
LIN {X 0,Y 509.505,Z 462.097,A -85,B 0,C 180,E1 -5482.27,E2 -5482.27} C_VEL
LIN {X 0,Y 509.313,Z 469.183,A -85,B 0,C 180,E1 -5483.661,E2 -5483.661} C_VEL
LIN {X 0,Y 509.248,Z 473.897,A -85,B 0,C 180,E1 -5484.853,E2 -5484.853} C_VEL
LIN {X 0,Y 509.247,Z 477.499,A -85,B 0,C 180,E1 -5486.043,E2 -5486.043} C_VEL
LIN {X 0,Y 509.202,Z 479.356,A -85,B 0,C 180,E1 -5486.835,E2 -5486.835} C_VEL
LIN {X 0,Y 509.162,Z 480.747,A -85,B 0,C 180,E1 -5487.626,E2 -5487.626} C_VEL
LIN {X 0,Y 509.074,Z 482.346,A -85,B 0,C 180,E1 -5489.208,E2 -5489.208} C_VEL
LIN {X 0,Y 509.067,Z 482.561,A -85,B 0,C 180,E1 -5489.999,E2 -5489.999} C_VEL
LIN {X 0,Y 509.113,Z 481.74,A -85,B 0,C 180,E1 -5491.581,E2 -5491.581} C_VEL
LIN {X 0,Y 509.162,Z 480.748,A -85,B 0,C 180,E1 -5492.373,E2 -5492.373} C_VEL
LIN {X 0,Y 509.202,Z 479.356,A -85,B 0,C 180,E1 -5493.164,E2 -5493.164} C_VEL
LIN {X 0,Y 509.206,Z 476.426,A -85,B 0,C 180,E1 -5494.353,E2 -5494.353} C_VEL
LIN {X 0,Y 509.312,Z 472.461,A -85,B 0,C 180,E1 -5495.542,E2 -5495.542} C_VEL
LIN {X 0,Y 509.366,Z 466.461,A -85,B 0,C 180,E1 -5496.914,E2 -5496.914} C_VEL
LIN {X 0,Y 509.561,Z 459.691,A -85,B 0,C 180,E1 -5498.126,E2 -5498.126} C_VEL
LIN {X 0,Y 509.77,Z 451.414,A -85,B 0,C 180,E1 -5499.322,E2 -5499.322} C_VEL
LIN {X 0,Y 510.033,Z 442.925,A -85,B 0,C 180,E1 -5500.319,E2 -5500.319} C_VEL
LIN {X 0,Y 510.4,Z 432.433,A -85,B 0,C 180,E1 -5501.315,E2 -5501.315} C_VEL
LIN {X 0,Y 510.697,Z 421.938,A -85,B 0,C 180,E1 -5502.121,E2 -5502.121} C_VEL
LIN {X 0,Y 511.061,Z 410.657,A -85,B 0,C 180,E1 -5502.811,E2 -5502.811} C_VEL
LIN {X 0,Y 511.337,Z 398.935,A -85,B 0,C 180,E1 -5503.36,E2 -5503.36} C_VEL
LIN {X 0,Y 511.594,Z 386.337,A -85,B 0,C 180,E1 -5503.783,E2 -5503.783} C_VEL
LIN {X 0,Y 511.784,Z 373.5,A -85,B 0,C 180,E1 -5504.056,E2 -5504.056} C_VEL
LIN {X 0,Y 512.172,Z 282.329,A -85,B 0,C 180,E1 -5505.349,E2 -5505.349} C_VEL
LIN {X 0,Y 510.281,Z 270.906,A -85,B 0,C 180,E1 -5505.584,E2 -5505.584} C_VEL
LIN {X 0,Y 510.298,Z 269.126,A -85,B 0,C 180,E1 -5505.808,E2 -5505.808} C_VEL
LIN {X 0,Y 510.718,Z 250.991,A -85,B 0,C 180,E1 -5508.867,E2 -5508.867} C_VEL
LIN {X 0,Y 511.262,Z 232.686,A -85,B 0,C 180,E1 -5511.998,E2 -5511.998} C_VEL
LIN {X 0,Y 510.465,Z 226.531,A -85,B 0,C 180,E1 -5513.108,E2 -5513.108} C_VEL
LIN {X 0,Y 509.887,Z 223.513,A -85,B 0,C 180,E1 -5513.721,E2 -5513.721} C_VEL
LIN {X 0,Y 509.88,Z 223.471,A -85,B 0,C 180,E1 -5517.055,E2 -5517.055} C_VEL
LIN {X 0,Y 509.86,Z 223.477,A -85,B 0,C 180,E1 -5519.75,E2 -5519.75} C_VEL
LIN {X 0,Y 509.876,Z 223.469,A -85,B 0,C 180,E1 -5522.773,E2 -5522.773} C_VEL
LIN {X 0,Y 509.825,Z 223.478,A -85,B 0,C 180,E1 -5525.576,E2 -5525.576} C_VEL
LIN {X 0,Y 509.85,Z 223.476,A -85,B 0,C 180,E1 -5528.337,E2 -5528.337} C_VEL
LIN {X 0,Y 509.845,Z 223.471,A -85,B 0,C 180,E1 -5531.425,E2 -5531.425} C_VEL
LIN {X 0,Y 509.841,Z 223.475,A -85,B 0,C 180,E1 -5534.668,E2 -5534.668} C_VEL
LIN {X 0,Y 509.847,Z 223.477,A -85,B 0,C 180,E1 -5538.103,E2 -5538.103} C_VEL
LIN {X 0,Y 509.833,Z 223.477,A -85,B 0,C 180,E1 -5540.644,E2 -5540.644} C_VEL
LIN {X 0,Y 509.808,Z 223.476,A -85,B 0,C 180,E1 -5543.644,E2 -5543.644} C_VEL
LIN {X 0,Y 509.838,Z 223.48,A -85,B 0,C 180,E1 -5546.536,E2 -5546.536} C_VEL
LIN {X 0,Y 509.832,Z 223.473,A -85,B 0,C 180,E1 -5549.331,E2 -5549.331} C_VEL
LIN {X 0,Y 509.831,Z 223.473,A -85,B 0,C 180,E1 -5552.049,E2 -5552.049} C_VEL
LIN {X 0,Y 509.8,Z 223.483,A -85,B 0,C 180,E1 -5554.698,E2 -5554.698} C_VEL
LIN {X 0,Y 509.822,Z 223.475,A -85,B 0,C 180,E1 -5557.457,E2 -5557.457} C_VEL
LIN {X 0,Y 509.904,Z 223.464,A -85,B 0,C 180,E1 -5559.842,E2 -5559.842} C_VEL
LIN {X 0,Y 509.853,Z 223.479,A -85,B 0,C 180,E1 -5563.171,E2 -5563.171} C_VEL
LIN {X 0,Y 509.838,Z 223.472,A -85,B 0,C 180,E1 -5565.631,E2 -5565.631} C_VEL
LIN {X 0,Y 509.9,Z 223.468,A -85,B 0,C 180,E1 -5568.872,E2 -5568.872} C_VEL
LIN {X 0,Y 509.879,Z 223.466,A -85,B 0,C 180,E1 -5572.075,E2 -5572.075} C_VEL
LIN {X 0,Y 509.954,Z 223.458,A -85,B 0,C 180,E1 -5574.461,E2 -5574.461} C_VEL
LIN {X 0,Y 510.027,Z 223.456,A -85,B 0,C 180,E1 -5577.628,E2 -5577.628} C_VEL
LIN {X 0,Y 510.016,Z 223.451,A -85,B 0,C 180,E1 -5579.997,E2 -5579.997} C_VEL
LIN {X 0,Y 510.023,Z 223.449,A -85,B 0,C 180,E1 -5582.366,E2 -5582.366} C_VEL
LIN {X 0,Y 509.916,Z 223.468,A -85,B 0,C 180,E1 -5585.534,E2 -5585.534} C_VEL
LIN {X 0,Y 509.86,Z 223.476,A -85,B 0,C 180,E1 -5587.92,E2 -5587.92} C_VEL
LIN {X 0,Y 509.847,Z 223.471,A -85,B 0,C 180,E1 -5591.124,E2 -5591.124} C_VEL
LIN {X 0,Y 509.829,Z 223.476,A -85,B 0,C 180,E1 -5593.55,E2 -5593.55} C_VEL
LIN {X 0,Y 509.823,Z 223.483,A -85,B 0,C 180,E1 -5596.001,E2 -5596.001} C_VEL
LIN {X 0,Y 509.819,Z 223.479,A -85,B 0,C 180,E1 -5598.482,E2 -5598.482} C_VEL
LIN {X 0,Y 509.83,Z 223.474,A -85,B 0,C 180,E1 -5600.999,E2 -5600.999} C_VEL
LIN {X 0,Y 509.8,Z 223.477,A -85,B 0,C 180,E1 -5603.561,E2 -5603.561} C_VEL
LIN {X 0,Y 509.861,Z 223.478,A -85,B 0,C 180,E1 -5606.369,E2 -5606.369} C_VEL
LIN {X 0,Y 509.834,Z 223.473,A -85,B 0,C 180,E1 -5609.724,E2 -5609.724} C_VEL
LIN {X 0,Y 509.847,Z 223.477,A -85,B 0,C 180,E1 -5612.771,E2 -5612.771} C_VEL
LIN {X 0,Y 509.815,Z 223.475,A -85,B 0,C 180,E1 -5615.578,E2 -5615.578} C_VEL
LIN {X 0,Y 509.824,Z 223.479,A -85,B 0,C 180,E1 -5618.335,E2 -5618.335} C_VEL
LIN {X 0,Y 509.836,Z 223.476,A -85,B 0,C 180,E1 -5621.422,E2 -5621.422} C_VEL
LIN {X 0,Y 509.826,Z 223.483,A -85,B 0,C 180,E1 -5624.666,E2 -5624.666} C_VEL
LIN {X 0,Y 509.913,Z 223.611,A -85,B 0,C 180,E1 -5625.396,E2 -5625.396} C_VEL
LIN {X 0,Y 510.733,Z 229.532,A -85,B 0,C 180,E1 -5626.527,E2 -5626.527} C_VEL
LIN {X 0,Y 510.49,Z 244.552,A -85,B 0,C 180,E1 -5629.211,E2 -5629.211} C_VEL
LIN {X 0,Y 510.255,Z 256.657,A -85,B 0,C 180,E1 -5631.35,E2 -5631.35} C_VEL
LIN {X 0,Y 509.767,Z 258.344,A -85,B 0,C 180,E1 -5631.456,E2 -5631.456} C_VEL
LIN {X 0,Y 506.544,Z 266.749,A -85,B 0,C 180,E1 -5631.491,E2 -5631.491} C_VEL
LIN {X 0,Y 505.172,Z 272.78,A -85,B 0,C 180,E1 -5631.512,E2 -5631.512} C_VEL
LIN {X 0,Y 504.96,Z 279.207,A -85,B 0,C 180,E1 -5631.592,E2 -5631.592} C_VEL
LIN {X 0,Y 505.274,Z 287.823,A -85,B 0,C 180,E1 -5631.758,E2 -5631.758} C_VEL
LIN {X 0,Y 504.838,Z 365.137,A -85,B 0,C 180,E1 -5632.887,E2 -5632.887} C_VEL
LIN {X 0,Y 504.636,Z 378.174,A -85,B 0,C 180,E1 -5633.239,E2 -5633.239} C_VEL
LIN {X 0,Y 504.367,Z 391.196,A -85,B 0,C 180,E1 -5633.763,E2 -5633.763} C_VEL
LIN {X 0,Y 504.051,Z 402.826,A -85,B 0,C 180,E1 -5634.401,E2 -5634.401} C_VEL
LIN {X 0,Y 503.604,Z 414.238,A -85,B 0,C 180,E1 -5635.204,E2 -5635.204} C_VEL
LIN {X 0,Y 503.281,Z 425.089,A -85,B 0,C 180,E1 -5636.164,E2 -5636.164} C_VEL
LIN {X 0,Y 502.928,Z 434.59,A -85,B 0,C 180,E1 -5637.215,E2 -5637.215} C_VEL
LIN {X 0,Y 502.686,Z 442.329,A -85,B 0,C 180,E1 -5638.26,E2 -5638.26} C_VEL
LIN {X 0,Y 502.444,Z 450.006,A -85,B 0,C 180,E1 -5639.533,E2 -5639.533} C_VEL
LIN {X 0,Y 502.275,Z 455.525,A -85,B 0,C 180,E1 -5640.678,E2 -5640.678} C_VEL
LIN {X 0,Y 502.166,Z 461.056,A -85,B 0,C 180,E1 -5642.166,E2 -5642.166} C_VEL
LIN {X 0,Y 502.098,Z 464.868,A -85,B 0,C 180,E1 -5643.604,E2 -5643.604} C_VEL
LIN {X 0,Y 501.987,Z 467.47,A -85,B 0,C 180,E1 -5645.166,E2 -5645.166} C_VEL
LIN {X 0,Y 501.991,Z 468.226,A -85,B 0,C 180,E1 -5646.047,E2 -5646.047} C_VEL
LIN {X 0,Y 501.975,Z 468.469,A -85,B 0,C 180,E1 -5647.513,E2 -5647.513} C_VEL
LIN {X 0,Y 501.957,Z 467.734,A -85,B 0,C 180,E1 -5648.653,E2 -5648.653} C_VEL
LIN {X 0,Y 502.046,Z 466.386,A -85,B 0,C 180,E1 -5649.691,E2 -5649.691} C_VEL
LIN {X 0,Y 502.129,Z 463.081,A -85,B 0,C 180,E1 -5651.222,E2 -5651.222} C_VEL
LIN {X 0,Y 502.189,Z 459.072,A -85,B 0,C 180,E1 -5652.508,E2 -5652.508} C_VEL
LIN {X 0,Y 502.338,Z 453.984,A -85,B 0,C 180,E1 -5653.752,E2 -5653.752} C_VEL
LIN {X 0,Y 502.526,Z 446.862,A -85,B 0,C 180,E1 -5655.112,E2 -5655.112} C_VEL
LIN {X 0,Y 502.791,Z 439.341,A -85,B 0,C 180,E1 -5656.254,E2 -5656.254} C_VEL
LIN {X 0,Y 503.101,Z 429.85,A -85,B 0,C 180,E1 -5657.424,E2 -5657.424} C_VEL
LIN {X 0,Y 503.415,Z 419.745,A -85,B 0,C 180,E1 -5658.424,E2 -5658.424} C_VEL
LIN {X 0,Y 503.821,Z 407.968,A -85,B 0,C 180,E1 -5659.35,E2 -5659.35} C_VEL
LIN {X 0,Y 504.218,Z 396.286,A -85,B 0,C 180,E1 -5660.068,E2 -5660.068} C_VEL
LIN {X 0,Y 504.493,Z 384.191,A -85,B 0,C 180,E1 -5660.63,E2 -5660.63} C_VEL
LIN {X 0,Y 504.75,Z 371.901,A -85,B 0,C 180,E1 -5661.039,E2 -5661.039} C_VEL
LIN {X 0,Y 504.944,Z 359.104,A -85,B 0,C 180,E1 -5661.307,E2 -5661.307} C_VEL
LIN {X 0,Y 505.235,Z 268.712,A -85,B 0,C 180,E1 -5662.609,E2 -5662.609} C_VEL
LIN {X 0,Y 503.276,Z 257.734,A -85,B 0,C 180,E1 -5662.856,E2 -5662.856} C_VEL
LIN {X 0,Y 503.523,Z 250.288,A -85,B 0,C 180,E1 -5664.193,E2 -5664.193} C_VEL
LIN {X 0,Y 504.035,Z 232.277,A -85,B 0,C 180,E1 -5667.603,E2 -5667.603} C_VEL
LIN {X 0,Y 503.008,Z 224.431,A -85,B 0,C 180,E1 -5669.2,E2 -5669.2} C_VEL
LIN {X 0,Y 502.871,Z 224.347,A -85,B 0,C 180,E1 -5671.602,E2 -5671.602} C_VEL
LIN {X 0,Y 502.867,Z 224.347,A -85,B 0,C 180,E1 -5673.205,E2 -5673.205} C_VEL
LIN {X 0,Y 502.869,Z 224.34,A -85,B 0,C 180,E1 -5676.42,E2 -5676.42} C_VEL
LIN {X 0,Y 502.836,Z 224.346,A -85,B 0,C 180,E1 -5678.845,E2 -5678.845} C_VEL
LIN {X 0,Y 502.856,Z 224.341,A -85,B 0,C 180,E1 -5682.102,E2 -5682.102} C_VEL
LIN {X 0,Y 502.812,Z 224.352,A -85,B 0,C 180,E1 -5685.401,E2 -5685.401} C_VEL
LIN {X 0,Y 502.81,Z 224.353,A -85,B 0,C 180,E1 -5688.124,E2 -5688.124} C_VEL
LIN {X 0,Y 502.794,Z 224.351,A -85,B 0,C 180,E1 -5690.538,E2 -5690.538} C_VEL
LIN {X 0,Y 502.753,Z 224.354,A -85,B 0,C 180,E1 -5693.043,E2 -5693.043} C_VEL
LIN {X 0,Y 502.767,Z 224.355,A -85,B 0,C 180,E1 -5695.68,E2 -5695.68} C_VEL
LIN {X 0,Y 502.764,Z 224.355,A -85,B 0,C 180,E1 -5698.378,E2 -5698.378} C_VEL
LIN {X 0,Y 502.764,Z 224.353,A -85,B 0,C 180,E1 -5701.146,E2 -5701.146} C_VEL
LIN {X 0,Y 502.758,Z 224.357,A -85,B 0,C 180,E1 -5703.998,E2 -5703.998} C_VEL
LIN {X 0,Y 502.722,Z 224.359,A -85,B 0,C 180,E1 -5707.176,E2 -5707.176} C_VEL
LIN {X 0,Y 502.743,Z 224.358,A -85,B 0,C 180,E1 -5710.02,E2 -5710.02} C_VEL
LIN {X 0,Y 502.724,Z 224.356,A -85,B 0,C 180,E1 -5713.237,E2 -5713.237} C_VEL
LIN {X 0,Y 502.754,Z 224.354,A -85,B 0,C 180,E1 -5715.663,E2 -5715.663} C_VEL
LIN {X 0,Y 502.743,Z 224.358,A -85,B 0,C 180,E1 -5719.016,E2 -5719.016} C_VEL
LIN {X 0,Y 502.771,Z 224.344,A -85,B 0,C 180,E1 -5722.049,E2 -5722.049} C_VEL
LIN {X 0,Y 502.776,Z 224.359,A -85,B 0,C 180,E1 -5725.037,E2 -5725.037} C_VEL
LIN {X 0,Y 502.762,Z 224.352,A -85,B 0,C 180,E1 -5727.918,E2 -5727.918} C_VEL
LIN {X 0,Y 502.777,Z 224.346,A -85,B 0,C 180,E1 -5730.713,E2 -5730.713} C_VEL
LIN {X 0,Y 502.759,Z 224.358,A -85,B 0,C 180,E1 -5733.464,E2 -5733.464} C_VEL
LIN {X 0,Y 502.754,Z 224.355,A -85,B 0,C 180,E1 -5736.088,E2 -5736.088} C_VEL
LIN {X 0,Y 502.774,Z 224.351,A -85,B 0,C 180,E1 -5738.692,E2 -5738.692} C_VEL
LIN {X 0,Y 502.803,Z 224.346,A -85,B 0,C 180,E1 -5741.251,E2 -5741.251} C_VEL
LIN {X 0,Y 502.832,Z 224.339,A -85,B 0,C 180,E1 -5744.667,E2 -5744.667} C_VEL
LIN {X 0,Y 502.866,Z 224.346,A -85,B 0,C 180,E1 -5748.046,E2 -5748.046} C_VEL
LIN {X 0,Y 502.844,Z 224.34,A -85,B 0,C 180,E1 -5751.159,E2 -5751.159} C_VEL
LIN {X 0,Y 502.87,Z 224.334,A -85,B 0,C 180,E1 -5753.584,E2 -5753.584} C_VEL
LIN {X 0,Y 502.835,Z 224.341,A -85,B 0,C 180,E1 -5756.798,E2 -5756.798} C_VEL
LIN {X 0,Y 502.898,Z 224.341,A -85,B 0,C 180,E1 -5758.401,E2 -5758.401} C_VEL
LIN {X 0,Y 502.971,Z 224.327,A -85,B 0,C 180,E1 -5760.803,E2 -5760.803} C_VEL
LIN {X 0,Y 503.009,Z 224.324,A -85,B 0,C 180,E1 -5762.405,E2 -5762.405} C_VEL
LIN {X 0,Y 502.904,Z 224.324,A -85,B 0,C 180,E1 -5765.616,E2 -5765.616} C_VEL
LIN {X 0,Y 502.875,Z 224.339,A -85,B 0,C 180,E1 -5768.036,E2 -5768.036} C_VEL
LIN {X 0,Y 502.878,Z 224.339,A -85,B 0,C 180,E1 -5771.286,E2 -5771.286} C_VEL
LIN {X 0,Y 502.834,Z 224.345,A -85,B 0,C 180,E1 -5774.573,E2 -5774.573} C_VEL
LIN {X 0,Y 502.817,Z 224.349,A -85,B 0,C 180,E1 -5777.071,E2 -5777.071} C_VEL
LIN {X 0,Y 502.826,Z 224.346,A -85,B 0,C 180,E1 -5779.602,E2 -5779.602} C_VEL
LIN {X 0,Y 502.81,Z 224.352,A -85,B 0,C 180,E1 -5782.703,E2 -5782.703} C_VEL
LIN {X 0,Y 502.797,Z 224.348,A -85,B 0,C 180,E1 -5785.68,E2 -5785.68} C_VEL
LIN {X 0,Y 502.782,Z 224.352,A -85,B 0,C 180,E1 -5788.378,E2 -5788.378} C_VEL
LIN {X 0,Y 502.8,Z 224.352,A -85,B 0,C 180,E1 -5791.145,E2 -5791.145} C_VEL
LIN {X 0,Y 502.795,Z 224.35,A -85,B 0,C 180,E1 -5793.997,E2 -5793.997} C_VEL
LIN {X 0,Y 502.773,Z 224.357,A -85,B 0,C 180,E1 -5797.177,E2 -5797.177} C_VEL
LIN {X 0,Y 502.782,Z 224.353,A -85,B 0,C 180,E1 -5800.018,E2 -5800.018} C_VEL
LIN {X 0,Y 502.781,Z 224.349,A -85,B 0,C 180,E1 -5802.196,E2 -5802.196} C_VEL
LIN {X 0,Y 502.796,Z 224.356,A -85,B 0,C 180,E1 -5805.471,E2 -5805.471} C_VEL
LIN {X 0,Y 502.79,Z 224.357,A -85,B 0,C 180,E1 -5807.86,E2 -5807.86} C_VEL
LIN {X 0,Y 502.802,Z 224.349,A -85,B 0,C 180,E1 -5811.024,E2 -5811.024} C_VEL
LIN {X 0,Y 502.78,Z 224.358,A -85,B 0,C 180,E1 -5814.17,E2 -5814.17} C_VEL
LIN {X 0,Y 502.842,Z 224.343,A -85,B 0,C 180,E1 -5816.994,E2 -5816.994} C_VEL
LIN {X 0,Y 502.823,Z 224.353,A -85,B 0,C 180,E1 -5820.066,E2 -5820.066} C_VEL
LIN {X 0,Y 502.832,Z 224.351,A -85,B 0,C 180,E1 -5822.533,E2 -5822.533} C_VEL
LIN {X 0,Y 502.841,Z 224.381,A -85,B 0,C 180,E1 -5826.006,E2 -5826.006} C_VEL
LIN {X 0,Y 503.947,Z 230.182,A -85,B 0,C 180,E1 -5827.161,E2 -5827.161} C_VEL
LIN {X 0,Y 504.35,Z 235.422,A -85,B 0,C 180,E1 -5828.114,E2 -5828.114} C_VEL
LIN {X 0,Y 503.724,Z 255.268,A -85,B 0,C 180,E1 -5831.578,E2 -5831.578} C_VEL
LIN {X 0,Y 503.283,Z 270.557,A -85,B 0,C 180,E1 -5834.174,E2 -5834.174} C_VEL
LIN {X 0,Y 504.772,Z 279.863,A -85,B 0,C 180,E1 -5834.386,E2 -5834.386} C_VEL
LIN {X 0,Y 505.397,Z 285.358,A -85,B 0,C 180,E1 -5834.485,E2 -5834.485} C_VEL
LIN {X 0,Y 504.875,Z 378.945,A -85,B 0,C 180,E1 -5835.849,E2 -5835.849} C_VEL
LIN {X 0,Y 504.601,Z 391.984,A -85,B 0,C 180,E1 -5836.201,E2 -5836.201} C_VEL
LIN {X 0,Y 504.286,Z 404.59,A -85,B 0,C 180,E1 -5836.705,E2 -5836.705} C_VEL
LIN {X 0,Y 503.949,Z 416.708,A -85,B 0,C 180,E1 -5837.37,E2 -5837.37} C_VEL
LIN {X 0,Y 503.596,Z 428.711,A -85,B 0,C 180,E1 -5838.223,E2 -5838.223} C_VEL
LIN {X 0,Y 503.184,Z 438.921,A -85,B 0,C 180,E1 -5839.131,E2 -5839.131} C_VEL
LIN {X 0,Y 502.875,Z 448.1,A -85,B 0,C 180,E1 -5840.142,E2 -5840.142} C_VEL
LIN {X 0,Y 502.6,Z 457.037,A -85,B 0,C 180,E1 -5841.354,E2 -5841.354} C_VEL
LIN {X 0,Y 502.36,Z 464.229,A -85,B 0,C 180,E1 -5842.564,E2 -5842.564} C_VEL
LIN {X 0,Y 502.241,Z 469.082,A -85,B 0,C 180,E1 -5843.572,E2 -5843.572} C_VEL
LIN {X 0,Y 502.181,Z 473.797,A -85,B 0,C 180,E1 -5844.78,E2 -5844.78} C_VEL
LIN {X 0,Y 502.14,Z 477.399,A -85,B 0,C 180,E1 -5845.987,E2 -5845.987} C_VEL
LIN {X 0,Y 502.122,Z 479.257,A -85,B 0,C 180,E1 -5846.79,E2 -5846.79} C_VEL
LIN {X 0,Y 502.037,Z 481.642,A -85,B 0,C 180,E1 -5848.395,E2 -5848.395} C_VEL
LIN {X 0,Y 501.981,Z 482.463,A -85,B 0,C 180,E1 -5849.999,E2 -5849.999} C_VEL
LIN {X 0,Y 502.036,Z 481.642,A -85,B 0,C 180,E1 -5851.604,E2 -5851.604} C_VEL
LIN {X 0,Y 502.066,Z 480.648,A -85,B 0,C 180,E1 -5852.406,E2 -5852.406} C_VEL
LIN {X 0,Y 502.122,Z 479.256,A -85,B 0,C 180,E1 -5853.209,E2 -5853.209} C_VEL
LIN {X 0,Y 502.104,Z 476.325,A -85,B 0,C 180,E1 -5854.415,E2 -5854.415} C_VEL
LIN {X 0,Y 502.229,Z 472.358,A -85,B 0,C 180,E1 -5855.621,E2 -5855.621} C_VEL
LIN {X 0,Y 502.292,Z 466.355,A -85,B 0,C 180,E1 -5857.011,E2 -5857.011} C_VEL
LIN {X 0,Y 502.493,Z 459.583,A -85,B 0,C 180,E1 -5858.242,E2 -5858.242} C_VEL
LIN {X 0,Y 502.742,Z 451.304,A -85,B 0,C 180,E1 -5859.453,E2 -5859.453} C_VEL
LIN {X 0,Y 503.019,Z 442.811,A -85,B 0,C 180,E1 -5860.464,E2 -5860.464} C_VEL
LIN {X 0,Y 503.439,Z 432.315,A -85,B 0,C 180,E1 -5861.474,E2 -5861.474} C_VEL
LIN {X 0,Y 503.717,Z 421.815,A -85,B 0,C 180,E1 -5862.292,E2 -5862.292} C_VEL
LIN {X 0,Y 504.124,Z 410.532,A -85,B 0,C 180,E1 -5862.99,E2 -5862.99} C_VEL
LIN {X 0,Y 504.426,Z 398.803,A -85,B 0,C 180,E1 -5863.546,E2 -5863.546} C_VEL
LIN {X 0,Y 504.739,Z 385.285,A -85,B 0,C 180,E1 -5864,E2 -5864} C_VEL
LIN {X 0,Y 504.925,Z 371.75,A -85,B 0,C 180,E1 -5864.277,E2 -5864.277} C_VEL
LIN {X 0,Y 505.359,Z 283.448,A -85,B 0,C 180,E1 -5865.544,E2 -5865.544} C_VEL
LIN {X 0,Y 503.287,Z 270.589,A -85,B 0,C 180,E1 -5865.821,E2 -5865.821} C_VEL
LIN {X 0,Y 503.37,Z 265.521,A -85,B 0,C 180,E1 -5866.631,E2 -5866.631} C_VEL
LIN {X 0,Y 503.799,Z 249.66,A -85,B 0,C 180,E1 -5869.348,E2 -5869.348} C_VEL
LIN {X 0,Y 504.329,Z 233.789,A -85,B 0,C 180,E1 -5872.101,E2 -5872.101} C_VEL
LIN {X 0,Y 503.229,Z 226.438,A -85,B 0,C 180,E1 -5873.454,E2 -5873.454} C_VEL
LIN {X 0,Y 502.843,Z 224.418,A -85,B 0,C 180,E1 -5873.883,E2 -5873.883} C_VEL
LIN {X 0,Y 502.841,Z 224.348,A -85,B 0,C 180,E1 -5876.566,E2 -5876.566} C_VEL
LIN {X 0,Y 502.826,Z 224.35,A -85,B 0,C 180,E1 -5879.287,E2 -5879.287} C_VEL
LIN {X 0,Y 502.786,Z 224.359,A -85,B 0,C 180,E1 -5882.083,E2 -5882.083} C_VEL
LIN {X 0,Y 502.8,Z 224.35,A -85,B 0,C 180,E1 -5884.965,E2 -5884.965} C_VEL
LIN {X 0,Y 502.793,Z 224.353,A -85,B 0,C 180,E1 -5888.484,E2 -5888.484} C_VEL
LIN {X 0,Y 502.779,Z 224.351,A -85,B 0,C 180,E1 -5891.069,E2 -5891.069} C_VEL
LIN {X 0,Y 502.758,Z 224.354,A -85,B 0,C 180,E1 -5893.371,E2 -5893.371} C_VEL
LIN {X 0,Y 502.78,Z 224.352,A -85,B 0,C 180,E1 -5895.658,E2 -5895.658} C_VEL
LIN {X 0,Y 502.796,Z 224.352,A -85,B 0,C 180,E1 -5897.859,E2 -5897.859} C_VEL
LIN {X 0,Y 502.793,Z 224.349,A -85,B 0,C 180,E1 -5901.021,E2 -5901.021} C_VEL
LIN {X 0,Y 502.77,Z 224.357,A -85,B 0,C 180,E1 -5904.168,E2 -5904.168} C_VEL
LIN {X 0,Y 502.803,Z 224.352,A -85,B 0,C 180,E1 -5906.997,E2 -5906.997} C_VEL
LIN {X 0,Y 502.809,Z 224.348,A -85,B 0,C 180,E1 -5910.064,E2 -5910.064} C_VEL
LIN {X 0,Y 502.772,Z 224.353,A -85,B 0,C 180,E1 -5913.458,E2 -5913.458} C_VEL
LIN {X 0,Y 502.764,Z 224.353,A -85,B 0,C 180,E1 -5916.083,E2 -5916.083} C_VEL
LIN {X 0,Y 502.776,Z 224.355,A -85,B 0,C 180,E1 -5918.686,E2 -5918.686} C_VEL
LIN {X 0,Y 502.815,Z 224.349,A -85,B 0,C 180,E1 -5921.245,E2 -5921.245} C_VEL
LIN {X 0,Y 502.844,Z 224.346,A -85,B 0,C 180,E1 -5924.598,E2 -5924.598} C_VEL
LIN {X 0,Y 502.871,Z 224.34,A -85,B 0,C 180,E1 -5928.037,E2 -5928.037} C_VEL
LIN {X 0,Y 502.83,Z 224.351,A -85,B 0,C 180,E1 -5931.153,E2 -5931.153} C_VEL
LIN {X 0,Y 502.879,Z 224.345,A -85,B 0,C 180,E1 -5933.578,E2 -5933.578} C_VEL
LIN {X 0,Y 502.82,Z 224.343,A -85,B 0,C 180,E1 -5936.792,E2 -5936.792} C_VEL
LIN {X 0,Y 502.877,Z 224.339,A -85,B 0,C 180,E1 -5938.396,E2 -5938.396} C_VEL
LIN {X 0,Y 502.985,Z 224.326,A -85,B 0,C 180,E1 -5939.997,E2 -5939.997} C_VEL
LIN {X 0,Y 502.991,Z 224.325,A -85,B 0,C 180,E1 -5942.4,E2 -5942.4} C_VEL
LIN {X 0,Y 502.871,Z 224.345,A -85,B 0,C 180,E1 -5945.611,E2 -5945.611} C_VEL
LIN {X 0,Y 502.832,Z 224.35,A -85,B 0,C 180,E1 -5948.031,E2 -5948.031} C_VEL
LIN {X 0,Y 502.822,Z 224.348,A -85,B 0,C 180,E1 -5951.281,E2 -5951.281} C_VEL
LIN {X 0,Y 502.814,Z 224.349,A -85,B 0,C 180,E1 -5954.568,E2 -5954.568} C_VEL
LIN {X 0,Y 502.78,Z 224.349,A -85,B 0,C 180,E1 -5957.067,E2 -5957.067} C_VEL
LIN {X 0,Y 502.8,Z 224.352,A -85,B 0,C 180,E1 -5959.597,E2 -5959.597} C_VEL
LIN {X 0,Y 502.782,Z 224.353,A -85,B 0,C 180,E1 -5962.699,E2 -5962.699} C_VEL
LIN {X 0,Y 502.779,Z 224.352,A -85,B 0,C 180,E1 -5965.675,E2 -5965.675} C_VEL
LIN {X 0,Y 502.775,Z 224.356,A -85,B 0,C 180,E1 -5968.373,E2 -5968.373} C_VEL
LIN {X 0,Y 502.769,Z 224.354,A -85,B 0,C 180,E1 -5971.141,E2 -5971.141} C_VEL
LIN {X 0,Y 502.781,Z 224.355,A -85,B 0,C 180,E1 -5973.991,E2 -5973.991} C_VEL
LIN {X 0,Y 502.753,Z 224.357,A -85,B 0,C 180,E1 -5977.176,E2 -5977.176} C_VEL
LIN {X 0,Y 502.793,Z 224.353,A -85,B 0,C 180,E1 -5980.009,E2 -5980.009} C_VEL
LIN {X 0,Y 502.8,Z 224.354,A -85,B 0,C 180,E1 -5982.2,E2 -5982.2} C_VEL
LIN {X 0,Y 502.866,Z 224.553,A -85,B 0,C 180,E1 -5985.266,E2 -5985.266} C_VEL
LIN {X 0,Y 503.795,Z 230.961,A -85,B 0,C 180,E1 -5986.497,E2 -5986.497} C_VEL
LIN {X 0,Y 503.472,Z 246.296,A -85,B 0,C 180,E1 -5989.264,E2 -5989.264} C_VEL
LIN {X 0,Y 503.304,Z 257.358,A -85,B 0,C 180,E1 -5991.213,E2 -5991.213} C_VEL
LIN {X 0,Y 504.142,Z 262.537,A -85,B 0,C 180,E1 -5991.352,E2 -5991.352} C_VEL
LIN {X 0,Y 505.392,Z 270.508,A -85,B 0,C 180,E1 -5991.509,E2 -5991.509} C_VEL
LIN {X 0,Y 505.274,Z 287.823,A -85,B 0,C 180,E1 -5991.758,E2 -5991.758} C_VEL
LIN {X 0,Y 504.582,Z 293.672,A -85,B 0,C 180,E1 -5991.821,E2 -5991.821} C_VEL
LIN {X 0,Y 498.881,Z 312.671,A -85,B 0,C 180,E1 -5991.92,E2 -5991.92} C_VEL
LIN {X 0,Y 498.303,Z 318.513,A -85,B 0,C 180,E1 -5991.988,E2 -5991.988} C_VEL
LIN {X 0,Y 497.96,Z 365.773,A -85,B 0,C 180,E1 -5992.7,E2 -5992.7} C_VEL
LIN {X 0,Y 497.71,Z 379.179,A -85,B 0,C 180,E1 -5993.075,E2 -5993.075} C_VEL
LIN {X 0,Y 497.442,Z 391.873,A -85,B 0,C 180,E1 -5993.603,E2 -5993.603} C_VEL
LIN {X 0,Y 497.044,Z 404.459,A -85,B 0,C 180,E1 -5994.321,E2 -5994.321} C_VEL
LIN {X 0,Y 496.587,Z 415.93,A -85,B 0,C 180,E1 -5995.162,E2 -5995.162} C_VEL
LIN {X 0,Y 496.249,Z 426.136,A -85,B 0,C 180,E1 -5996.108,E2 -5996.108} C_VEL
LIN {X 0,Y 495.886,Z 435.56,A -85,B 0,C 180,E1 -5997.185,E2 -5997.185} C_VEL
LIN {X 0,Y 495.593,Z 443.874,A -85,B 0,C 180,E1 -5998.353,E2 -5998.353} C_VEL
LIN {X 0,Y 495.372,Z 451.248,A -85,B 0,C 180,E1 -5999.649,E2 -5999.649} C_VEL
LIN {X 0,Y 495.202,Z 456.046,A -85,B 0,C 180,E1 -6000.685,E2 -6000.685} C_VEL
LIN {X 0,Y 495.089,Z 461.065,A -85,B 0,C 180,E1 -6002.067,E2 -6002.067} C_VEL
LIN {X 0,Y 495.01,Z 464.689,A -85,B 0,C 180,E1 -6003.428,E2 -6003.428} C_VEL
LIN {X 0,Y 494.921,Z 467.107,A -85,B 0,C 180,E1 -6004.787,E2 -6004.787} C_VEL
LIN {X 0,Y 494.879,Z 468.098,A -85,B 0,C 180,E1 -6005.68,E2 -6005.68} C_VEL
LIN {X 0,Y 494.862,Z 468.569,A -85,B 0,C 180,E1 -6006.569,E2 -6006.569} C_VEL
LIN {X 0,Y 494.886,Z 468.58,A -85,B 0,C 180,E1 -6007.454,E2 -6007.454} C_VEL
LIN {X 0,Y 494.855,Z 468.158,A -85,B 0,C 180,E1 -6008.331,E2 -6008.331} C_VEL
LIN {X 0,Y 494.924,Z 466.723,A -85,B 0,C 180,E1 -6009.575,E2 -6009.575} C_VEL
LIN {X 0,Y 495.021,Z 464.056,A -85,B 0,C 180,E1 -6010.942,E2 -6010.942} C_VEL
LIN {X 0,Y 495.094,Z 460.059,A -85,B 0,C 180,E1 -6012.33,E2 -6012.33} C_VEL
LIN {X 0,Y 495.214,Z 455.566,A -85,B 0,C 180,E1 -6013.512,E2 -6013.512} C_VEL
LIN {X 0,Y 495.382,Z 449.791,A -85,B 0,C 180,E1 -6014.717,E2 -6014.717} C_VEL
LIN {X 0,Y 495.655,Z 441.761,A -85,B 0,C 180,E1 -6016.052,E2 -6016.052} C_VEL
LIN {X 0,Y 495.941,Z 433.942,A -85,B 0,C 180,E1 -6017.104,E2 -6017.104} C_VEL
LIN {X 0,Y 496.316,Z 424.079,A -85,B 0,C 180,E1 -6018.184,E2 -6018.184} C_VEL
LIN {X 0,Y 496.682,Z 413.805,A -85,B 0,C 180,E1 -6019.091,E2 -6019.091} C_VEL
LIN {X 0,Y 497.144,Z 401.962,A -85,B 0,C 180,E1 -6019.925,E2 -6019.925} C_VEL
LIN {X 0,Y 497.434,Z 390.531,A -85,B 0,C 180,E1 -6020.547,E2 -6020.547} C_VEL
LIN {X 0,Y 497.741,Z 377.581,A -85,B 0,C 180,E1 -6021.066,E2 -6021.066} C_VEL
LIN {X 0,Y 497.962,Z 364.728,A -85,B 0,C 180,E1 -6021.41,E2 -6021.41} C_VEL
LIN {X 0,Y 498.411,Z 269.388,A -85,B 0,C 180,E1 -6022.817,E2 -6022.817} C_VEL
LIN {X 0,Y 496.337,Z 258.066,A -85,B 0,C 180,E1 -6023.071,E2 -6023.071} C_VEL
LIN {X 0,Y 496.336,Z 256.381,A -85,B 0,C 180,E1 -6023.296,E2 -6023.296} C_VEL
LIN {X 0,Y 496.776,Z 241.439,A -85,B 0,C 180,E1 -6026.148,E2 -6026.148} C_VEL
LIN {X 0,Y 496.968,Z 231.997,A -85,B 0,C 180,E1 -6027.975,E2 -6027.975} C_VEL
LIN {X 0,Y 496.013,Z 225.533,A -85,B 0,C 180,E1 -6029.29,E2 -6029.29} C_VEL
LIN {X 0,Y 495.955,Z 225.202,A -85,B 0,C 180,E1 -6029.595,E2 -6029.595} C_VEL
LIN {X 0,Y 495.954,Z 225.205,A -85,B 0,C 180,E1 -6032.437,E2 -6032.437} C_VEL
LIN {X 0,Y 495.869,Z 225.218,A -85,B 0,C 180,E1 -6035.694,E2 -6035.694} C_VEL
LIN {X 0,Y 495.835,Z 225.219,A -85,B 0,C 180,E1 -6038.149,E2 -6038.149} C_VEL
LIN {X 0,Y 495.83,Z 225.224,A -85,B 0,C 180,E1 -6041.446,E2 -6041.446} C_VEL
LIN {X 0,Y 495.751,Z 225.227,A -85,B 0,C 180,E1 -6044.785,E2 -6044.785} C_VEL
LIN {X 0,Y 495.762,Z 225.23,A -85,B 0,C 180,E1 -6048.173,E2 -6048.173} C_VEL
LIN {X 0,Y 495.739,Z 225.228,A -85,B 0,C 180,E1 -6050.758,E2 -6050.758} C_VEL
LIN {X 0,Y 495.708,Z 225.233,A -85,B 0,C 180,E1 -6053.39,E2 -6053.39} C_VEL
LIN {X 0,Y 495.728,Z 225.237,A -85,B 0,C 180,E1 -6056.072,E2 -6056.072} C_VEL
LIN {X 0,Y 495.711,Z 225.228,A -85,B 0,C 180,E1 -6058.819,E2 -6058.819} C_VEL
LIN {X 0,Y 495.724,Z 225.232,A -85,B 0,C 180,E1 -6061.728,E2 -6061.728} C_VEL
LIN {X 0,Y 495.729,Z 225.228,A -85,B 0,C 180,E1 -6064.695,E2 -6064.695} C_VEL
LIN {X 0,Y 495.678,Z 225.235,A -85,B 0,C 180,E1 -6067.567,E2 -6067.567} C_VEL
LIN {X 0,Y 495.715,Z 225.233,A -85,B 0,C 180,E1 -6070.048,E2 -6070.048} C_VEL
LIN {X 0,Y 495.678,Z 225.237,A -85,B 0,C 180,E1 -6072.889,E2 -6072.889} C_VEL
LIN {X 0,Y 495.699,Z 225.233,A -85,B 0,C 180,E1 -6076.001,E2 -6076.001} C_VEL
LIN {X 0,Y 495.706,Z 225.23,A -85,B 0,C 180,E1 -6079.299,E2 -6079.299} C_VEL
LIN {X 0,Y 495.725,Z 225.224,A -85,B 0,C 180,E1 -6081.411,E2 -6081.411} C_VEL
LIN {X 0,Y 495.728,Z 225.229,A -85,B 0,C 180,E1 -6084.465,E2 -6084.465} C_VEL
LIN {X 0,Y 495.734,Z 225.232,A -85,B 0,C 180,E1 -6087.408,E2 -6087.408} C_VEL
LIN {X 0,Y 495.726,Z 225.221,A -85,B 0,C 180,E1 -6090.255,E2 -6090.255} C_VEL
LIN {X 0,Y 495.724,Z 225.23,A -85,B 0,C 180,E1 -6093.274,E2 -6093.274} C_VEL
LIN {X 0,Y 495.728,Z 225.23,A -85,B 0,C 180,E1 -6096.616,E2 -6096.616} C_VEL
LIN {X 0,Y 495.771,Z 225.229,A -85,B 0,C 180,E1 -6099.328,E2 -6099.328} C_VEL
LIN {X 0,Y 495.772,Z 225.216,A -85,B 0,C 180,E1 -6101.832,E2 -6101.832} C_VEL
LIN {X 0,Y 495.775,Z 225.22,A -85,B 0,C 180,E1 -6105.22,E2 -6105.22} C_VEL
LIN {X 0,Y 495.817,Z 225.218,A -85,B 0,C 180,E1 -6108.557,E2 -6108.557} C_VEL
LIN {X 0,Y 495.811,Z 225.221,A -85,B 0,C 180,E1 -6111.854,E2 -6111.854} C_VEL
LIN {X 0,Y 495.853,Z 225.208,A -85,B 0,C 180,E1 -6114.309,E2 -6114.309} C_VEL
LIN {X 0,Y 495.975,Z 225.197,A -85,B 0,C 180,E1 -6117.566,E2 -6117.566} C_VEL
LIN {X 0,Y 495.924,Z 225.205,A -85,B 0,C 180,E1 -6120.815,E2 -6120.815} C_VEL
LIN {X 0,Y 495.976,Z 225.199,A -85,B 0,C 180,E1 -6122.439,E2 -6122.439} C_VEL
LIN {X 0,Y 495.864,Z 225.201,A -85,B 0,C 180,E1 -6125.696,E2 -6125.696} C_VEL
LIN {X 0,Y 495.832,Z 225.217,A -85,B 0,C 180,E1 -6128.151,E2 -6128.151} C_VEL
LIN {X 0,Y 495.854,Z 225.213,A -85,B 0,C 180,E1 -6131.448,E2 -6131.448} C_VEL
LIN {X 0,Y 495.785,Z 225.22,A -85,B 0,C 180,E1 -6134.785,E2 -6134.785} C_VEL
LIN {X 0,Y 495.763,Z 225.225,A -85,B 0,C 180,E1 -6137.322,E2 -6137.322} C_VEL
LIN {X 0,Y 495.774,Z 225.224,A -85,B 0,C 180,E1 -6139.892,E2 -6139.892} C_VEL
LIN {X 0,Y 495.766,Z 225.227,A -85,B 0,C 180,E1 -6142.862,E2 -6142.862} C_VEL
LIN {X 0,Y 495.753,Z 225.224,A -85,B 0,C 180,E1 -6146.072,E2 -6146.072} C_VEL
LIN {X 0,Y 495.737,Z 225.234,A -85,B 0,C 180,E1 -6148.819,E2 -6148.819} C_VEL
LIN {X 0,Y 495.762,Z 225.224,A -85,B 0,C 180,E1 -6151.726,E2 -6151.726} C_VEL
LIN {X 0,Y 495.768,Z 225.227,A -85,B 0,C 180,E1 -6154.693,E2 -6154.693} C_VEL
LIN {X 0,Y 495.73,Z 225.233,A -85,B 0,C 180,E1 -6157.564,E2 -6157.564} C_VEL
LIN {X 0,Y 495.755,Z 225.228,A -85,B 0,C 180,E1 -6160.046,E2 -6160.046} C_VEL
LIN {X 0,Y 495.713,Z 225.229,A -85,B 0,C 180,E1 -6162.886,E2 -6162.886} C_VEL
LIN {X 0,Y 495.733,Z 225.232,A -85,B 0,C 180,E1 -6165.998,E2 -6165.998} C_VEL
LIN {X 0,Y 495.74,Z 225.231,A -85,B 0,C 180,E1 -6169.297,E2 -6169.297} C_VEL
LIN {X 0,Y 495.755,Z 225.23,A -85,B 0,C 180,E1 -6171.408,E2 -6171.408} C_VEL
LIN {X 0,Y 495.754,Z 225.23,A -85,B 0,C 180,E1 -6174.462,E2 -6174.462} C_VEL
LIN {X 0,Y 495.777,Z 225.225,A -85,B 0,C 180,E1 -6177.406,E2 -6177.406} C_VEL
LIN {X 0,Y 495.774,Z 225.233,A -85,B 0,C 180,E1 -6180.254,E2 -6180.254} C_VEL
LIN {X 0,Y 495.815,Z 225.221,A -85,B 0,C 180,E1 -6183.255,E2 -6183.255} C_VEL
LIN {X 0,Y 495.835,Z 225.415,A -85,B 0,C 180,E1 -6185.896,E2 -6185.896} C_VEL
LIN {X 0,Y 497.371,Z 234.124,A -85,B 0,C 180,E1 -6187.572,E2 -6187.572} C_VEL
LIN {X 0,Y 497.19,Z 242.229,A -85,B 0,C 180,E1 -6189.023,E2 -6189.023} C_VEL
LIN {X 0,Y 496.627,Z 259.517,A -85,B 0,C 180,E1 -6192.073,E2 -6192.073} C_VEL
LIN {X 0,Y 496.306,Z 270.451,A -85,B 0,C 180,E1 -6193.946,E2 -6193.946} C_VEL
LIN {X 0,Y 497.699,Z 279.169,A -85,B 0,C 180,E1 -6194.152,E2 -6194.152} C_VEL
LIN {X 0,Y 498.547,Z 285.338,A -85,B 0,C 180,E1 -6194.27,E2 -6194.27} C_VEL
LIN {X 0,Y 498.014,Z 378.738,A -85,B 0,C 180,E1 -6195.65,E2 -6195.65} C_VEL
LIN {X 0,Y 497.718,Z 391.815,A -85,B 0,C 180,E1 -6196.006,E2 -6196.006} C_VEL
LIN {X 0,Y 497.373,Z 404.441,A -85,B 0,C 180,E1 -6196.517,E2 -6196.517} C_VEL
LIN {X 0,Y 497.053,Z 415.518,A -85,B 0,C 180,E1 -6197.122,E2 -6197.122} C_VEL
LIN {X 0,Y 496.704,Z 426,A -85,B 0,C 180,E1 -6197.85,E2 -6197.85} C_VEL
LIN {X 0,Y 496.298,Z 436.684,A -85,B 0,C 180,E1 -6198.772,E2 -6198.772} C_VEL
LIN {X 0,Y 495.916,Z 446.306,A -85,B 0,C 180,E1 -6199.796,E2 -6199.796} C_VEL
LIN {X 0,Y 495.613,Z 454.192,A -85,B 0,C 180,E1 -6200.82,E2 -6200.82} C_VEL
LIN {X 0,Y 495.372,Z 461.891,A -85,B 0,C 180,E1 -6202.048,E2 -6202.048} C_VEL
LIN {X 0,Y 495.17,Z 468.98,A -85,B 0,C 180,E1 -6203.48,E2 -6203.48} C_VEL
LIN {X 0,Y 495.115,Z 473.697,A -85,B 0,C 180,E1 -6204.705,E2 -6204.705} C_VEL
LIN {X 0,Y 495.034,Z 477.3,A -85,B 0,C 180,E1 -6205.929,E2 -6205.929} C_VEL
LIN {X 0,Y 495.043,Z 479.158,A -85,B 0,C 180,E1 -6206.744,E2 -6206.744} C_VEL
LIN {X 0,Y 494.962,Z 481.544,A -85,B 0,C 180,E1 -6208.372,E2 -6208.372} C_VEL
LIN {X 0,Y 494.9,Z 482.365,A -85,B 0,C 180,E1 -6209.999,E2 -6209.999} C_VEL
LIN {X 0,Y 494.962,Z 481.543,A -85,B 0,C 180,E1 -6211.627,E2 -6211.627} C_VEL
LIN {X 0,Y 495.043,Z 479.156,A -85,B 0,C 180,E1 -6213.255,E2 -6213.255} C_VEL
LIN {X 0,Y 495.009,Z 476.223,A -85,B 0,C 180,E1 -6214.478,E2 -6214.478} C_VEL
LIN {X 0,Y 495.146,Z 472.255,A -85,B 0,C 180,E1 -6215.701,E2 -6215.701} C_VEL
LIN {X 0,Y 495.242,Z 466.149,A -85,B 0,C 180,E1 -6217.132,E2 -6217.132} C_VEL
LIN {X 0,Y 495.452,Z 459.477,A -85,B 0,C 180,E1 -6218.359,E2 -6218.359} C_VEL
LIN {X 0,Y 495.726,Z 451.197,A -85,B 0,C 180,E1 -6219.588,E2 -6219.588} C_VEL
LIN {X 0,Y 496.004,Z 442.703,A -85,B 0,C 180,E1 -6220.614,E2 -6220.614} C_VEL
LIN {X 0,Y 496.475,Z 432.207,A -85,B 0,C 180,E1 -6221.637,E2 -6221.637} C_VEL
LIN {X 0,Y 496.781,Z 420.762,A -85,B 0,C 180,E1 -6222.535,E2 -6222.535} C_VEL
LIN {X 0,Y 497.231,Z 408.481,A -85,B 0,C 180,E1 -6223.278,E2 -6223.278} C_VEL
LIN {X 0,Y 497.577,Z 396.089,A -85,B 0,C 180,E1 -6223.84,E2 -6223.84} C_VEL
LIN {X 0,Y 497.924,Z 383.328,A -85,B 0,C 180,E1 -6224.247,E2 -6224.247} C_VEL
LIN {X 0,Y 498.047,Z 369.848,A -85,B 0,C 180,E1 -6224.505,E2 -6224.505} C_VEL
LIN {X 0,Y 498.422,Z 283.301,A -85,B 0,C 180,E1 -6225.767,E2 -6225.767} C_VEL
LIN {X 0,Y 496.316,Z 270.488,A -85,B 0,C 180,E1 -6226.053,E2 -6226.053} C_VEL
LIN {X 0,Y 496.432,Z 264.206,A -85,B 0,C 180,E1 -6227.082,E2 -6227.082} C_VEL
LIN {X 0,Y 496.934,Z 247.11,A -85,B 0,C 180,E1 -6230.056,E2 -6230.056} C_VEL
LIN {X 0,Y 497.389,Z 234.892,A -85,B 0,C 180,E1 -6232.207,E2 -6232.207} C_VEL
LIN {X 0,Y 495.896,Z 225.713,A -85,B 0,C 180,E1 -6233.933,E2 -6233.933} C_VEL
LIN {X 0,Y 495.794,Z 225.229,A -85,B 0,C 180,E1 -6234.161,E2 -6234.161} C_VEL
LIN {X 0,Y 495.788,Z 225.227,A -85,B 0,C 180,E1 -6236.975,E2 -6236.975} C_VEL
LIN {X 0,Y 495.769,Z 225.232,A -85,B 0,C 180,E1 -6239.745,E2 -6239.745} C_VEL
LIN {X 0,Y 495.771,Z 225.227,A -85,B 0,C 180,E1 -6242.593,E2 -6242.593} C_VEL
LIN {X 0,Y 495.748,Z 225.232,A -85,B 0,C 180,E1 -6245.537,E2 -6245.537} C_VEL
LIN {X 0,Y 495.76,Z 225.227,A -85,B 0,C 180,E1 -6248.766,E2 -6248.766} C_VEL
LIN {X 0,Y 495.747,Z 225.23,A -85,B 0,C 180,E1 -6251.781,E2 -6251.781} C_VEL
LIN {X 0,Y 495.739,Z 225.229,A -85,B 0,C 180,E1 -6255.139,E2 -6255.139} C_VEL
LIN {X 0,Y 495.746,Z 225.235,A -85,B 0,C 180,E1 -6258.216,E2 -6258.216} C_VEL
LIN {X 0,Y 495.746,Z 225.226,A -85,B 0,C 180,E1 -6261.406,E2 -6261.406} C_VEL
LIN {X 0,Y 495.743,Z 225.235,A -85,B 0,C 180,E1 -6264.46,E2 -6264.46} C_VEL
LIN {X 0,Y 495.751,Z 225.227,A -85,B 0,C 180,E1 -6267.402,E2 -6267.402} C_VEL
LIN {X 0,Y 495.756,Z 225.229,A -85,B 0,C 180,E1 -6270.251,E2 -6270.251} C_VEL
LIN {X 0,Y 495.737,Z 225.231,A -85,B 0,C 180,E1 -6273.268,E2 -6273.268} C_VEL
LIN {X 0,Y 495.736,Z 225.233,A -85,B 0,C 180,E1 -6276.61,E2 -6276.61} C_VEL
LIN {X 0,Y 495.776,Z 225.228,A -85,B 0,C 180,E1 -6279.322,E2 -6279.322} C_VEL
LIN {X 0,Y 495.776,Z 225.221,A -85,B 0,C 180,E1 -6281.826,E2 -6281.826} C_VEL
LIN {X 0,Y 495.771,Z 225.23,A -85,B 0,C 180,E1 -6285.214,E2 -6285.214} C_VEL
LIN {X 0,Y 495.842,Z 225.216,A -85,B 0,C 180,E1 -6288.552,E2 -6288.552} C_VEL
LIN {X 0,Y 495.808,Z 225.22,A -85,B 0,C 180,E1 -6291.848,E2 -6291.848} C_VEL
LIN {X 0,Y 495.865,Z 225.213,A -85,B 0,C 180,E1 -6294.304,E2 -6294.304} C_VEL
LIN {X 0,Y 495.962,Z 225.207,A -85,B 0,C 180,E1 -6297.561,E2 -6297.561} C_VEL
LIN {X 0,Y 495.955,Z 225.202,A -85,B 0,C 180,E1 -6299.997,E2 -6299.997} C_VEL
LIN {X 0,Y 495.959,Z 225.201,A -85,B 0,C 180,E1 -6302.434,E2 -6302.434} C_VEL
LIN {X 0,Y 495.829,Z 225.222,A -85,B 0,C 180,E1 -6305.691,E2 -6305.691} C_VEL
LIN {X 0,Y 495.796,Z 225.225,A -85,B 0,C 180,E1 -6308.146,E2 -6308.146} C_VEL
LIN {X 0,Y 495.806,Z 225.223,A -85,B 0,C 180,E1 -6311.443,E2 -6311.443} C_VEL
LIN {X 0,Y 495.763,Z 225.227,A -85,B 0,C 180,E1 -6314.78,E2 -6314.78} C_VEL
LIN {X 0,Y 495.761,Z 225.235,A -85,B 0,C 180,E1 -6318.169,E2 -6318.169} C_VEL
LIN {X 0,Y 495.755,Z 225.228,A -85,B 0,C 180,E1 -6320.754,E2 -6320.754} C_VEL
LIN {X 0,Y 495.721,Z 225.23,A -85,B 0,C 180,E1 -6323.385,E2 -6323.385} C_VEL
LIN {X 0,Y 495.739,Z 225.234,A -85,B 0,C 180,E1 -6326.067,E2 -6326.067} C_VEL
LIN {X 0,Y 495.722,Z 225.233,A -85,B 0,C 180,E1 -6328.814,E2 -6328.814} C_VEL
LIN {X 0,Y 495.729,Z 225.23,A -85,B 0,C 180,E1 -6331.722,E2 -6331.722} C_VEL
LIN {X 0,Y 495.75,Z 225.232,A -85,B 0,C 180,E1 -6334.692,E2 -6334.692} C_VEL
LIN {X 0,Y 495.704,Z 225.233,A -85,B 0,C 180,E1 -6337.559,E2 -6337.559} C_VEL
LIN {X 0,Y 495.751,Z 225.235,A -85,B 0,C 180,E1 -6340.696,E2 -6340.696} C_VEL
LIN {X 0,Y 495.705,Z 225.239,A -85,B 0,C 180,E1 -6343.693,E2 -6343.693} C_VEL
LIN {X 0,Y 495.794,Z 225.278,A -85,B 0,C 180,E1 -6345.044,E2 -6345.044} C_VEL
LIN {X 0,Y 496.769,Z 230.843,A -85,B 0,C 180,E1 -6346.174,E2 -6346.174} C_VEL
LIN {X 0,Y 496.611,Z 242.516,A -85,B 0,C 180,E1 -6348.308,E2 -6348.308} C_VEL
LIN {X 0,Y 496.314,Z 257.574,A -85,B 0,C 180,E1 -6350.995,E2 -6350.995} C_VEL
LIN {X 0,Y 498.517,Z 270.117,A -85,B 0,C 180,E1 -6351.281,E2 -6351.281} C_VEL
LIN {X 0,Y 498.303,Z 318.513,A -85,B 0,C 180,E1 -6351.988,E2 -6351.988} C_VEL
LIN {X 0,Y 497.747,Z 324.348,A -85,B 0,C 180,E1 -6352.057,E2 -6352.057} C_VEL
LIN {X 0,Y 492.09,Z 343.338,A -85,B 0,C 180,E1 -6352.163,E2 -6352.163} C_VEL
LIN {X 0,Y 491.285,Z 349.184,A -85,B 0,C 180,E1 -6352.225,E2 -6352.225} C_VEL
LIN {X 0,Y 491.101,Z 367.829,A -85,B 0,C 180,E1 -6352.541,E2 -6352.541} C_VEL
LIN {X 0,Y 490.824,Z 380.092,A -85,B 0,C 180,E1 -6352.903,E2 -6352.903} C_VEL
LIN {X 0,Y 490.527,Z 392.177,A -85,B 0,C 180,E1 -6353.422,E2 -6353.422} C_VEL
LIN {X 0,Y 490.121,Z 404.267,A -85,B 0,C 180,E1 -6354.119,E2 -6354.119} C_VEL
LIN {X 0,Y 489.64,Z 415.669,A -85,B 0,C 180,E1 -6354.962,E2 -6354.962} C_VEL
LIN {X 0,Y 489.282,Z 426.06,A -85,B 0,C 180,E1 -6355.932,E2 -6355.932} C_VEL
LIN {X 0,Y 488.92,Z 434.484,A -85,B 0,C 180,E1 -6356.892,E2 -6356.892} C_VEL
LIN {X 0,Y 488.591,Z 442.877,A -85,B 0,C 180,E1 -6358.059,E2 -6358.059} C_VEL
LIN {X 0,Y 488.327,Z 449.997,A -85,B 0,C 180,E1 -6359.277,E2 -6359.277} C_VEL
LIN {X 0,Y 488.205,Z 454.542,A -85,B 0,C 180,E1 -6360.223,E2 -6360.223} C_VEL
LIN {X 0,Y 488.006,Z 459.975,A -85,B 0,C 180,E1 -6361.626,E2 -6361.626} C_VEL
LIN {X 0,Y 487.97,Z 462.804,A -85,B 0,C 180,E1 -6362.557,E2 -6362.557} C_VEL
LIN {X 0,Y 487.915,Z 465.013,A -85,B 0,C 180,E1 -6363.48,E2 -6363.48} C_VEL
LIN {X 0,Y 487.839,Z 466.713,A -85,B 0,C 180,E1 -6364.394,E2 -6364.394} C_VEL
LIN {X 0,Y 487.812,Z 467.854,A -85,B 0,C 180,E1 -6365.305,E2 -6365.305} C_VEL
LIN {X 0,Y 487.757,Z 468.534,A -85,B 0,C 180,E1 -6366.207,E2 -6366.207} C_VEL
LIN {X 0,Y 487.771,Z 468.724,A -85,B 0,C 180,E1 -6367.229,E2 -6367.229} C_VEL
LIN {X 0,Y 487.771,Z 467.746,A -85,B 0,C 180,E1 -6368.888,E2 -6368.888} C_VEL
LIN {X 0,Y 487.846,Z 466.569,A -85,B 0,C 180,E1 -6369.773,E2 -6369.773} C_VEL
LIN {X 0,Y 487.953,Z 463.917,A -85,B 0,C 180,E1 -6371.092,E2 -6371.092} C_VEL
LIN {X 0,Y 488.008,Z 460.183,A -85,B 0,C 180,E1 -6372.397,E2 -6372.397} C_VEL
LIN {X 0,Y 488.15,Z 455.26,A -85,B 0,C 180,E1 -6373.696,E2 -6373.696} C_VEL
LIN {X 0,Y 488.359,Z 449.021,A -85,B 0,C 180,E1 -6374.988,E2 -6374.988} C_VEL
LIN {X 0,Y 488.654,Z 441.255,A -85,B 0,C 180,E1 -6376.273,E2 -6376.273} C_VEL
LIN {X 0,Y 488.979,Z 433.296,A -85,B 0,C 180,E1 -6377.34,E2 -6377.34} C_VEL
LIN {X 0,Y 489.33,Z 423.579,A -85,B 0,C 180,E1 -6378.401,E2 -6378.401} C_VEL
LIN {X 0,Y 489.774,Z 412.76,A -85,B 0,C 180,E1 -6379.354,E2 -6379.354} C_VEL
LIN {X 0,Y 490.222,Z 402.258,A -85,B 0,C 180,E1 -6380.095,E2 -6380.095} C_VEL
LIN {X 0,Y 490.536,Z 390.902,A -85,B 0,C 180,E1 -6380.725,E2 -6380.725} C_VEL
LIN {X 0,Y 490.863,Z 377.853,A -85,B 0,C 180,E1 -6381.257,E2 -6381.257} C_VEL
LIN {X 0,Y 491.106,Z 364.492,A -85,B 0,C 180,E1 -6381.62,E2 -6381.62} C_VEL
LIN {X 0,Y 491.649,Z 270.572,A -85,B 0,C 180,E1 -6383.022,E2 -6383.022} C_VEL
LIN {X 0,Y 489.397,Z 258.204,A -85,B 0,C 180,E1 -6383.3,E2 -6383.3} C_VEL
LIN {X 0,Y 489.359,Z 257.229,A -85,B 0,C 180,E1 -6383.403,E2 -6383.403} C_VEL
LIN {X 0,Y 489.878,Z 241.106,A -85,B 0,C 180,E1 -6386.505,E2 -6386.505} C_VEL
LIN {X 0,Y 490.085,Z 233.749,A -85,B 0,C 180,E1 -6387.946,E2 -6387.946} C_VEL
LIN {X 0,Y 488.951,Z 226.187,A -85,B 0,C 180,E1 -6389.537,E2 -6389.537} C_VEL
LIN {X 0,Y 488.922,Z 226.082,A -85,B 0,C 180,E1 -6392.472,E2 -6392.472} C_VEL
LIN {X 0,Y 488.825,Z 226.095,A -85,B 0,C 180,E1 -6395.777,E2 -6395.777} C_VEL
LIN {X 0,Y 488.779,Z 226.097,A -85,B 0,C 180,E1 -6398.268,E2 -6398.268} C_VEL
LIN {X 0,Y 488.792,Z 226.101,A -85,B 0,C 180,E1 -6401.613,E2 -6401.613} C_VEL
LIN {X 0,Y 488.724,Z 226.103,A -85,B 0,C 180,E1 -6405.002,E2 -6405.002} C_VEL
LIN {X 0,Y 488.72,Z 226.104,A -85,B 0,C 180,E1 -6408.444,E2 -6408.444} C_VEL
LIN {X 0,Y 488.672,Z 226.108,A -85,B 0,C 180,E1 -6411.073,E2 -6411.073} C_VEL
LIN {X 0,Y 488.641,Z 226.117,A -85,B 0,C 180,E1 -6413.749,E2 -6413.749} C_VEL
LIN {X 0,Y 488.685,Z 226.112,A -85,B 0,C 180,E1 -6416.477,E2 -6416.477} C_VEL
LIN {X 0,Y 488.678,Z 226.103,A -85,B 0,C 180,E1 -6419.274,E2 -6419.274} C_VEL
LIN {X 0,Y 488.667,Z 226.116,A -85,B 0,C 180,E1 -6422.15,E2 -6422.15} C_VEL
LIN {X 0,Y 488.681,Z 226.102,A -85,B 0,C 180,E1 -6425.119,E2 -6425.119} C_VEL
LIN {X 0,Y 488.63,Z 226.118,A -85,B 0,C 180,E1 -6428.205,E2 -6428.205} C_VEL
LIN {X 0,Y 488.667,Z 226.115,A -85,B 0,C 180,E1 -6430.344,E2 -6430.344} C_VEL
LIN {X 0,Y 488.649,Z 226.106,A -85,B 0,C 180,E1 -6433.659,E2 -6433.659} C_VEL
LIN {X 0,Y 488.65,Z 226.114,A -85,B 0,C 180,E1 -6436.347,E2 -6436.347} C_VEL
LIN {X 0,Y 488.682,Z 226.102,A -85,B 0,C 180,E1 -6439.677,E2 -6439.677} C_VEL
LIN {X 0,Y 488.659,Z 226.109,A -85,B 0,C 180,E1 -6442.844,E2 -6442.844} C_VEL
LIN {X 0,Y 488.703,Z 226.105,A -85,B 0,C 180,E1 -6445.89,E2 -6445.89} C_VEL
LIN {X 0,Y 488.667,Z 226.111,A -85,B 0,C 180,E1 -6448.823,E2 -6448.823} C_VEL
LIN {X 0,Y 488.678,Z 226.102,A -85,B 0,C 180,E1 -6451.671,E2 -6451.671} C_VEL
LIN {X 0,Y 488.684,Z 226.107,A -85,B 0,C 180,E1 -6454.963,E2 -6454.963} C_VEL
LIN {X 0,Y 488.688,Z 226.107,A -85,B 0,C 180,E1 -6458.047,E2 -6458.047} C_VEL
LIN {X 0,Y 488.727,Z 226.095,A -85,B 0,C 180,E1 -6460.69,E2 -6460.69} C_VEL
LIN {X 0,Y 488.751,Z 226.095,A -85,B 0,C 180,E1 -6464.148,E2 -6464.148} C_VEL
LIN {X 0,Y 488.733,Z 226.105,A -85,B 0,C 180,E1 -6467.547,E2 -6467.547} C_VEL
LIN {X 0,Y 488.735,Z 226.103,A -85,B 0,C 180,E1 -6470.067,E2 -6470.067} C_VEL
LIN {X 0,Y 488.818,Z 226.08,A -85,B 0,C 180,E1 -6472.772,E2 -6472.772} C_VEL
LIN {X 0,Y 488.788,Z 226.083,A -85,B 0,C 180,E1 -6475.054,E2 -6475.054} C_VEL
LIN {X 0,Y 488.941,Z 226.073,A -85,B 0,C 180,E1 -6477.531,E2 -6477.531} C_VEL
LIN {X 0,Y 488.876,Z 226.083,A -85,B 0,C 180,E1 -6480.826,E2 -6480.826} C_VEL
LIN {X 0,Y 488.943,Z 226.074,A -85,B 0,C 180,E1 -6482.474,E2 -6482.474} C_VEL
LIN {X 0,Y 488.825,Z 226.078,A -85,B 0,C 180,E1 -6485.779,E2 -6485.779} C_VEL
LIN {X 0,Y 488.777,Z 226.098,A -85,B 0,C 180,E1 -6488.27,E2 -6488.27} C_VEL
LIN {X 0,Y 488.81,Z 226.091,A -85,B 0,C 180,E1 -6491.615,E2 -6491.615} C_VEL
LIN {X 0,Y 488.761,Z 226.092,A -85,B 0,C 180,E1 -6495.003,E2 -6495.003} C_VEL
LIN {X 0,Y 488.753,Z 226.1,A -85,B 0,C 180,E1 -6498.444,E2 -6498.444} C_VEL
LIN {X 0,Y 488.715,Z 226.107,A -85,B 0,C 180,E1 -6501.073,E2 -6501.073} C_VEL
LIN {X 0,Y 488.678,Z 226.099,A -85,B 0,C 180,E1 -6503.748,E2 -6503.748} C_VEL
LIN {X 0,Y 488.732,Z 226.107,A -85,B 0,C 180,E1 -6506.929,E2 -6506.929} C_VEL
LIN {X 0,Y 488.712,Z 226.101,A -85,B 0,C 180,E1 -6510.363,E2 -6510.363} C_VEL
LIN {X 0,Y 488.719,Z 226.109,A -85,B 0,C 180,E1 -6513.481,E2 -6513.481} C_VEL
LIN {X 0,Y 488.682,Z 226.106,A -85,B 0,C 180,E1 -6516.354,E2 -6516.354} C_VEL
LIN {X 0,Y 488.703,Z 226.109,A -85,B 0,C 180,E1 -6519.256,E2 -6519.256} C_VEL
LIN {X 0,Y 488.676,Z 226.104,A -85,B 0,C 180,E1 -6522.529,E2 -6522.529} C_VEL
LIN {X 0,Y 488.711,Z 226.107,A -85,B 0,C 180,E1 -6525.198,E2 -6525.198} C_VEL
LIN {X 0,Y 488.681,Z 226.108,A -85,B 0,C 180,E1 -6528.581,E2 -6528.581} C_VEL
LIN {X 0,Y 488.707,Z 226.105,A -85,B 0,C 180,E1 -6530.949,E2 -6530.949} C_VEL
LIN {X 0,Y 488.678,Z 226.116,A -85,B 0,C 180,E1 -6533.868,E2 -6533.868} C_VEL
LIN {X 0,Y 488.748,Z 226.099,A -85,B 0,C 180,E1 -6536.877,E2 -6536.877} C_VEL
LIN {X 0,Y 488.731,Z 226.105,A -85,B 0,C 180,E1 -6539.781,E2 -6539.781} C_VEL
LIN {X 0,Y 488.739,Z 226.106,A -85,B 0,C 180,E1 -6542.602,E2 -6542.602} C_VEL
LIN {X 0,Y 488.783,Z 226.253,A -85,B 0,C 180,E1 -6545.695,E2 -6545.695} C_VEL
LIN {X 0,Y 490.496,Z 236.458,A -85,B 0,C 180,E1 -6547.684,E2 -6547.684} C_VEL
LIN {X 0,Y 489.853,Z 253.372,A -85,B 0,C 180,E1 -6550.732,E2 -6550.732} C_VEL
LIN {X 0,Y 489.339,Z 270.15,A -85,B 0,C 180,E1 -6553.693,E2 -6553.693} C_VEL
LIN {X 0,Y 489.789,Z 273.535,A -85,B 0,C 180,E1 -6553.809,E2 -6553.809} C_VEL
LIN {X 0,Y 491.688,Z 285.341,A -85,B 0,C 180,E1 -6554.048,E2 -6554.048} C_VEL
LIN {X 0,Y 491.134,Z 378.528,A -85,B 0,C 180,E1 -6555.444,E2 -6555.444} C_VEL
LIN {X 0,Y 490.849,Z 391.641,A -85,B 0,C 180,E1 -6555.806,E2 -6555.806} C_VEL
LIN {X 0,Y 490.456,Z 404.286,A -85,B 0,C 180,E1 -6556.323,E2 -6556.323} C_VEL
LIN {X 0,Y 490.114,Z 415.68,A -85,B 0,C 180,E1 -6556.957,E2 -6556.957} C_VEL
LIN {X 0,Y 489.7,Z 427.164,A -85,B 0,C 180,E1 -6557.778,E2 -6557.778} C_VEL
LIN {X 0,Y 489.278,Z 437.632,A -85,B 0,C 180,E1 -6558.713,E2 -6558.713} C_VEL
LIN {X 0,Y 488.877,Z 446.186,A -85,B 0,C 180,E1 -6559.647,E2 -6559.647} C_VEL
LIN {X 0,Y 488.565,Z 454.077,A -85,B 0,C 180,E1 -6560.686,E2 -6560.686} C_VEL
LIN {X 0,Y 488.325,Z 461.782,A -85,B 0,C 180,E1 -6561.933,E2 -6561.933} C_VEL
LIN {X 0,Y 488.103,Z 468.875,A -85,B 0,C 180,E1 -6563.385,E2 -6563.385} C_VEL
LIN {X 0,Y 488.049,Z 473.595,A -85,B 0,C 180,E1 -6564.629,E2 -6564.629} C_VEL
LIN {X 0,Y 487.93,Z 477.198,A -85,B 0,C 180,E1 -6565.869,E2 -6565.869} C_VEL
LIN {X 0,Y 487.966,Z 479.059,A -85,B 0,C 180,E1 -6566.697,E2 -6566.697} C_VEL
LIN {X 0,Y 487.89,Z 481.446,A -85,B 0,C 180,E1 -6568.348,E2 -6568.348} C_VEL
LIN {X 0,Y 487.821,Z 482.267,A -85,B 0,C 180,E1 -6569.999,E2 -6569.999} C_VEL
LIN {X 0,Y 487.89,Z 481.445,A -85,B 0,C 180,E1 -6571.65,E2 -6571.65} C_VEL
LIN {X 0,Y 487.966,Z 479.057,A -85,B 0,C 180,E1 -6573.302,E2 -6573.302} C_VEL
LIN {X 0,Y 487.922,Z 476.124,A -85,B 0,C 180,E1 -6574.543,E2 -6574.543} C_VEL
LIN {X 0,Y 488.064,Z 472.156,A -85,B 0,C 180,E1 -6575.784,E2 -6575.784} C_VEL
LIN {X 0,Y 488.132,Z 467.047,A -85,B 0,C 180,E1 -6577.029,E2 -6577.029} C_VEL
LIN {X 0,Y 488.343,Z 460.611,A -85,B 0,C 180,E1 -6578.274,E2 -6578.274} C_VEL
LIN {X 0,Y 488.621,Z 452.584,A -85,B 0,C 180,E1 -6579.52,E2 -6579.52} C_VEL
LIN {X 0,Y 488.941,Z 444.402,A -85,B 0,C 180,E1 -6580.559,E2 -6580.559} C_VEL
LIN {X 0,Y 489.377,Z 434.422,A -85,B 0,C 180,E1 -6581.598,E2 -6581.598} C_VEL
LIN {X 0,Y 489.749,Z 424.565,A -85,B 0,C 180,E1 -6582.43,E2 -6582.43} C_VEL
LIN {X 0,Y 490.143,Z 414.018,A -85,B 0,C 180,E1 -6583.147,E2 -6583.147} C_VEL
LIN {X 0,Y 490.518,Z 402.083,A -85,B 0,C 180,E1 -6583.779,E2 -6583.779} C_VEL
LIN {X 0,Y 490.904,Z 389.454,A -85,B 0,C 180,E1 -6584.27,E2 -6584.27} C_VEL
LIN {X 0,Y 491.12,Z 377.552,A -85,B 0,C 180,E1 -6584.581,E2 -6584.581} C_VEL
LIN {X 0,Y 491.618,Z 284.283,A -85,B 0,C 180,E1 -6585.978,E2 -6585.978} C_VEL
LIN {X 0,Y 489.358,Z 270.385,A -85,B 0,C 180,E1 -6586.291,E2 -6586.291} C_VEL
LIN {X 0,Y 489.415,Z 265.333,A -85,B 0,C 180,E1 -6587.119,E2 -6587.119} C_VEL
LIN {X 0,Y 489.955,Z 248.231,A -85,B 0,C 180,E1 -6590.136,E2 -6590.136} C_VEL
LIN {X 0,Y 490.444,Z 236.005,A -85,B 0,C 180,E1 -6592.317,E2 -6592.317} C_VEL
LIN {X 0,Y 489,Z 227.414,A -85,B 0,C 180,E1 -6593.954,E2 -6593.954} C_VEL
LIN {X 0,Y 488.746,Z 226.136,A -85,B 0,C 180,E1 -6594.277,E2 -6594.277} C_VEL
LIN {X 0,Y 488.735,Z 226.107,A -85,B 0,C 180,E1 -6597.396,E2 -6597.396} C_VEL
LIN {X 0,Y 488.712,Z 226.109,A -85,B 0,C 180,E1 -6600.361,E2 -6600.361} C_VEL
LIN {X 0,Y 488.738,Z 226.105,A -85,B 0,C 180,E1 -6603.483,E2 -6603.483} C_VEL
LIN {X 0,Y 488.676,Z 226.111,A -85,B 0,C 180,E1 -6606.351,E2 -6606.351} C_VEL
LIN {X 0,Y 488.696,Z 226.106,A -85,B 0,C 180,E1 -6609.253,E2 -6609.253} C_VEL
LIN {X 0,Y 488.689,Z 226.111,A -85,B 0,C 180,E1 -6612.524,E2 -6612.524} C_VEL
LIN {X 0,Y 488.703,Z 226.105,A -85,B 0,C 180,E1 -6615.196,E2 -6615.196} C_VEL
LIN {X 0,Y 488.682,Z 226.114,A -85,B 0,C 180,E1 -6618.58,E2 -6618.58} C_VEL
LIN {X 0,Y 488.675,Z 226.107,A -85,B 0,C 180,E1 -6621.797,E2 -6621.797} C_VEL
LIN {X 0,Y 488.718,Z 226.105,A -85,B 0,C 180,E1 -6625.052,E2 -6625.052} C_VEL
LIN {X 0,Y 488.7,Z 226.106,A -85,B 0,C 180,E1 -6628.045,E2 -6628.045} C_VEL
LIN {X 0,Y 488.699,Z 226.114,A -85,B 0,C 180,E1 -6630.726,E2 -6630.726} C_VEL
LIN {X 0,Y 488.681,Z 226.108,A -85,B 0,C 180,E1 -6633.521,E2 -6633.521} C_VEL
LIN {X 0,Y 488.667,Z 226.11,A -85,B 0,C 180,E1 -6636.251,E2 -6636.251} C_VEL
LIN {X 0,Y 488.744,Z 226.106,A -85,B 0,C 180,E1 -6639.173,E2 -6639.173} C_VEL
LIN {X 0,Y 488.744,Z 226.098,A -85,B 0,C 180,E1 -6641.63,E2 -6641.63} C_VEL
LIN {X 0,Y 488.748,Z 226.107,A -85,B 0,C 180,E1 -6644.997,E2 -6644.997} C_VEL
LIN {X 0,Y 488.798,Z 226.093,A -85,B 0,C 180,E1 -6648.385,E2 -6648.385} C_VEL
LIN {X 0,Y 488.754,Z 226.1,A -85,B 0,C 180,E1 -6651.73,E2 -6651.73} C_VEL
LIN {X 0,Y 488.824,Z 226.09,A -85,B 0,C 180,E1 -6654.221,E2 -6654.221} C_VEL
LIN {X 0,Y 488.929,Z 226.083,A -85,B 0,C 180,E1 -6657.526,E2 -6657.526} C_VEL
LIN {X 0,Y 488.925,Z 226.078,A -85,B 0,C 180,E1 -6659.997,E2 -6659.997} C_VEL
LIN {X 0,Y 488.925,Z 226.077,A -85,B 0,C 180,E1 -6662.469,E2 -6662.469} C_VEL
LIN {X 0,Y 488.789,Z 226.099,A -85,B 0,C 180,E1 -6665.774,E2 -6665.774} C_VEL
LIN {X 0,Y 488.742,Z 226.102,A -85,B 0,C 180,E1 -6668.265,E2 -6668.265} C_VEL
LIN {X 0,Y 488.769,Z 226.102,A -85,B 0,C 180,E1 -6671.61,E2 -6671.61} C_VEL
LIN {X 0,Y 488.739,Z 226.101,A -85,B 0,C 180,E1 -6674.998,E2 -6674.998} C_VEL
LIN {X 0,Y 488.726,Z 226.107,A -85,B 0,C 180,E1 -6678.44,E2 -6678.44} C_VEL
LIN {X 0,Y 488.688,Z 226.107,A -85,B 0,C 180,E1 -6681.068,E2 -6681.068} C_VEL
LIN {X 0,Y 488.654,Z 226.113,A -85,B 0,C 180,E1 -6683.744,E2 -6683.744} C_VEL
LIN {X 0,Y 488.696,Z 226.113,A -85,B 0,C 180,E1 -6686.471,E2 -6686.471} C_VEL
LIN {X 0,Y 488.687,Z 226.106,A -85,B 0,C 180,E1 -6689.268,E2 -6689.268} C_VEL
LIN {X 0,Y 488.677,Z 226.112,A -85,B 0,C 180,E1 -6692.144,E2 -6692.144} C_VEL
LIN {X 0,Y 488.696,Z 226.109,A -85,B 0,C 180,E1 -6695.112,E2 -6695.112} C_VEL
LIN {X 0,Y 488.655,Z 226.115,A -85,B 0,C 180,E1 -6698.197,E2 -6698.197} C_VEL
LIN {X 0,Y 488.721,Z 226.109,A -85,B 0,C 180,E1 -6700.347,E2 -6700.347} C_VEL
LIN {X 0,Y 488.687,Z 226.113,A -85,B 0,C 180,E1 -6703.649,E2 -6703.649} C_VEL
LIN {X 0,Y 488.741,Z 226.178,A -85,B 0,C 180,E1 -6704.88,E2 -6704.88} C_VEL
LIN {X 0,Y 489.63,Z 230.861,A -85,B 0,C 180,E1 -6705.858,E2 -6705.858} C_VEL
LIN {X 0,Y 489.837,Z 237.092,A -85,B 0,C 180,E1 -6707.025,E2 -6707.025} C_VEL
LIN {X 0,Y 489.367,Z 253.329,A -85,B 0,C 180,E1 -6710.01,E2 -6710.01} C_VEL
LIN {X 0,Y 489.349,Z 257.683,A -85,B 0,C 180,E1 -6710.761,E2 -6710.761} C_VEL
LIN {X 0,Y 491.735,Z 271.22,A -85,B 0,C 180,E1 -6711.07,E2 -6711.07} C_VEL
LIN {X 0,Y 491.285,Z 349.184,A -85,B 0,C 180,E1 -6712.225,E2 -6712.225} C_VEL
LIN {X 0,Y 490.482,Z 355.021,A -85,B 0,C 180,E1 -6712.285,E2 -6712.285} C_VEL
LIN {X 0,Y 487.579,Z 364.489,A -85,B 0,C 180,E1 -6712.356,E2 -6712.356} C_VEL
LIN {X 0,Y 484.72,Z 373.864,A -85,B 0,C 180,E1 -6712.508,E2 -6712.508} C_VEL
LIN {X 0,Y 483.978,Z 379.543,A -85,B 0,C 180,E1 -6712.677,E2 -6712.677} C_VEL
LIN {X 0,Y 483.634,Z 392.342,A -85,B 0,C 180,E1 -6713.227,E2 -6713.227} C_VEL
LIN {X 0,Y 483.232,Z 404.094,A -85,B 0,C 180,E1 -6713.914,E2 -6713.914} C_VEL
LIN {X 0,Y 482.693,Z 415.724,A -85,B 0,C 180,E1 -6714.782,E2 -6714.782} C_VEL
LIN {X 0,Y 482.316,Z 425.608,A -85,B 0,C 180,E1 -6715.71,E2 -6715.71} C_VEL
LIN {X 0,Y 481.899,Z 435.377,A -85,B 0,C 180,E1 -6716.847,E2 -6716.847} C_VEL
LIN {X 0,Y 481.526,Z 443.811,A -85,B 0,C 180,E1 -6718.056,E2 -6718.056} C_VEL
LIN {X 0,Y 481.275,Z 450.633,A -85,B 0,C 180,E1 -6719.264,E2 -6719.264} C_VEL
LIN {X 0,Y 481.022,Z 457.018,A -85,B 0,C 180,E1 -6720.696,E2 -6720.696} C_VEL
LIN {X 0,Y 480.895,Z 461.851,A -85,B 0,C 180,E1 -6722.118,E2 -6722.118} C_VEL
LIN {X 0,Y 480.854,Z 464.33,A -85,B 0,C 180,E1 -6723.059,E2 -6723.059} C_VEL
LIN {X 0,Y 480.761,Z 466.189,A -85,B 0,C 180,E1 -6723.989,E2 -6723.989} C_VEL
LIN {X 0,Y 480.704,Z 467.688,A -85,B 0,C 180,E1 -6725.009,E2 -6725.009} C_VEL
LIN {X 0,Y 480.668,Z 468.427,A -85,B 0,C 180,E1 -6725.834,E2 -6725.834} C_VEL
LIN {X 0,Y 480.682,Z 468.85,A -85,B 0,C 180,E1 -6727.078,E2 -6727.078} C_VEL
LIN {X 0,Y 480.668,Z 468.182,A -85,B 0,C 180,E1 -6728.561,E2 -6728.561} C_VEL
LIN {X 0,Y 480.752,Z 467.167,A -85,B 0,C 180,E1 -6729.462,E2 -6729.462} C_VEL
LIN {X 0,Y 480.767,Z 465.729,A -85,B 0,C 180,E1 -6730.354,E2 -6730.354} C_VEL
LIN {X 0,Y 480.872,Z 462.367,A -85,B 0,C 180,E1 -6731.787,E2 -6731.787} C_VEL
LIN {X 0,Y 480.987,Z 458.451,A -85,B 0,C 180,E1 -6733.009,E2 -6733.009} C_VEL
LIN {X 0,Y 481.239,Z 452.01,A -85,B 0,C 180,E1 -6734.532,E2 -6734.532} C_VEL
LIN {X 0,Y 481.48,Z 444.895,A -85,B 0,C 180,E1 -6735.849,E2 -6735.849} C_VEL
LIN {X 0,Y 481.762,Z 437.677,A -85,B 0,C 180,E1 -6736.932,E2 -6736.932} C_VEL
LIN {X 0,Y 482.196,Z 428.251,A -85,B 0,C 180,E1 -6738.084,E2 -6738.084} C_VEL
LIN {X 0,Y 482.623,Z 418.105,A -85,B 0,C 180,E1 -6739.088,E2 -6739.088} C_VEL
LIN {X 0,Y 483.089,Z 407.343,A -85,B 0,C 180,E1 -6739.947,E2 -6739.947} C_VEL
LIN {X 0,Y 483.538,Z 395.316,A -85,B 0,C 180,E1 -6740.695,E2 -6740.695} C_VEL
LIN {X 0,Y 483.814,Z 383.508,A -85,B 0,C 180,E1 -6741.255,E2 -6741.255} C_VEL
LIN {X 0,Y 484.194,Z 370.719,A -85,B 0,C 180,E1 -6741.681,E2 -6741.681} C_VEL
LIN {X 0,Y 484.341,Z 357.697,A -85,B 0,C 180,E1 -6741.946,E2 -6741.946} C_VEL
LIN {X 0,Y 484.746,Z 270.974,A -85,B 0,C 180,E1 -6743.249,E2 -6743.249} C_VEL
LIN {X 0,Y 482.425,Z 258.196,A -85,B 0,C 180,E1 -6743.544,E2 -6743.544} C_VEL
LIN {X 0,Y 482.416,Z 256.781,A -85,B 0,C 180,E1 -6743.728,E2 -6743.728} C_VEL
LIN {X 0,Y 483.001,Z 239.718,A -85,B 0,C 180,E1 -6747.082,E2 -6747.082} C_VEL
LIN {X 0,Y 483.031,Z 234.503,A -85,B 0,C 180,E1 -6748.125,E2 -6748.125} C_VEL
LIN {X 0,Y 481.919,Z 227.129,A -85,B 0,C 180,E1 -6749.687,E2 -6749.687} C_VEL
LIN {X 0,Y 481.89,Z 226.958,A -85,B 0,C 180,E1 -6752.508,E2 -6752.508} C_VEL
LIN {X 0,Y 481.783,Z 226.971,A -85,B 0,C 180,E1 -6755.861,E2 -6755.861} C_VEL
LIN {X 0,Y 481.725,Z 226.976,A -85,B 0,C 180,E1 -6758.39,E2 -6758.39} C_VEL
LIN {X 0,Y 481.757,Z 226.974,A -85,B 0,C 180,E1 -6761.785,E2 -6761.785} C_VEL
LIN {X 0,Y 481.705,Z 226.979,A -85,B 0,C 180,E1 -6765.226,E2 -6765.226} C_VEL
LIN {X 0,Y 481.677,Z 226.98,A -85,B 0,C 180,E1 -6768.724,E2 -6768.724} C_VEL
LIN {X 0,Y 481.61,Z 226.99,A -85,B 0,C 180,E1 -6771.397,E2 -6771.397} C_VEL
LIN {X 0,Y 481.623,Z 226.991,A -85,B 0,C 180,E1 -6774.117,E2 -6774.117} C_VEL
LIN {X 0,Y 481.662,Z 226.982,A -85,B 0,C 180,E1 -6777.129,E2 -6777.129} C_VEL
LIN {X 0,Y 481.641,Z 226.981,A -85,B 0,C 180,E1 -6779.744,E2 -6779.744} C_VEL
LIN {X 0,Y 481.622,Z 226.99,A -85,B 0,C 180,E1 -6782.679,E2 -6782.679} C_VEL
LIN {X 0,Y 481.597,Z 226.984,A -85,B 0,C 180,E1 -6785.713,E2 -6785.713} C_VEL
LIN {X 0,Y 481.628,Z 226.991,A -85,B 0,C 180,E1 -6788.864,E2 -6788.864} C_VEL
LIN {X 0,Y 481.598,Z 226.987,A -85,B 0,C 180,E1 -6792.167,E2 -6792.167} C_VEL
LIN {X 0,Y 481.63,Z 226.986,A -85,B 0,C 180,E1 -6795.545,E2 -6795.545} C_VEL
LIN {X 0,Y 481.602,Z 226.991,A -85,B 0,C 180,E1 -6798.958,E2 -6798.958} C_VEL
LIN {X 0,Y 481.632,Z 226.976,A -85,B 0,C 180,E1 -6801.997,E2 -6801.997} C_VEL
LIN {X 0,Y 481.666,Z 226.987,A -85,B 0,C 180,E1 -6805.321,E2 -6805.321} C_VEL
LIN {X 0,Y 481.622,Z 226.984,A -85,B 0,C 180,E1 -6808.314,E2 -6808.314} C_VEL
LIN {X 0,Y 481.64,Z 226.979,A -85,B 0,C 180,E1 -6811.219,E2 -6811.219} C_VEL
LIN {X 0,Y 481.613,Z 226.986,A -85,B 0,C 180,E1 -6814.042,E2 -6814.042} C_VEL
LIN {X 0,Y 481.643,Z 226.985,A -85,B 0,C 180,E1 -6816.821,E2 -6816.821} C_VEL
LIN {X 0,Y 481.686,Z 226.982,A -85,B 0,C 180,E1 -6819.506,E2 -6819.506} C_VEL
LIN {X 0,Y 481.675,Z 226.966,A -85,B 0,C 180,E1 -6822.161,E2 -6822.161} C_VEL
LIN {X 0,Y 481.733,Z 226.966,A -85,B 0,C 180,E1 -6824.779,E2 -6824.779} C_VEL
LIN {X 0,Y 481.731,Z 226.976,A -85,B 0,C 180,E1 -6828.218,E2 -6828.218} C_VEL
LIN {X 0,Y 481.717,Z 226.976,A -85,B 0,C 180,E1 -6831.614,E2 -6831.614} C_VEL
LIN {X 0,Y 481.774,Z 226.96,A -85,B 0,C 180,E1 -6834.142,E2 -6834.142} C_VEL
LIN {X 0,Y 481.907,Z 226.949,A -85,B 0,C 180,E1 -6837.495,E2 -6837.495} C_VEL
LIN {X 0,Y 481.91,Z 226.957,A -85,B 0,C 180,E1 -6840.003,E2 -6840.003} C_VEL
LIN {X 0,Y 481.908,Z 226.95,A -85,B 0,C 180,E1 -6842.51,E2 -6842.51} C_VEL
LIN {X 0,Y 481.788,Z 226.955,A -85,B 0,C 180,E1 -6845.863,E2 -6845.863} C_VEL
LIN {X 0,Y 481.731,Z 226.977,A -85,B 0,C 180,E1 -6848.391,E2 -6848.391} C_VEL
LIN {X 0,Y 481.756,Z 226.97,A -85,B 0,C 180,E1 -6851.787,E2 -6851.787} C_VEL
LIN {X 0,Y 481.746,Z 226.963,A -85,B 0,C 180,E1 -6855.227,E2 -6855.227} C_VEL
LIN {X 0,Y 481.715,Z 226.981,A -85,B 0,C 180,E1 -6858.724,E2 -6858.724} C_VEL
LIN {X 0,Y 481.653,Z 226.983,A -85,B 0,C 180,E1 -6861.397,E2 -6861.397} C_VEL
LIN {X 0,Y 481.657,Z 226.973,A -85,B 0,C 180,E1 -6864.116,E2 -6864.116} C_VEL
LIN {X 0,Y 481.7,Z 226.986,A -85,B 0,C 180,E1 -6867.128,E2 -6867.128} C_VEL
LIN {X 0,Y 481.675,Z 226.979,A -85,B 0,C 180,E1 -6869.743,E2 -6869.743} C_VEL
LIN {X 0,Y 481.661,Z 226.98,A -85,B 0,C 180,E1 -6872.677,E2 -6872.677} C_VEL
LIN {X 0,Y 481.64,Z 226.987,A -85,B 0,C 180,E1 -6875.711,E2 -6875.711} C_VEL
LIN {X 0,Y 481.675,Z 226.98,A -85,B 0,C 180,E1 -6878.861,E2 -6878.861} C_VEL
LIN {X 0,Y 481.639,Z 226.982,A -85,B 0,C 180,E1 -6882.164,E2 -6882.164} C_VEL
LIN {X 0,Y 481.664,Z 226.99,A -85,B 0,C 180,E1 -6885.543,E2 -6885.543} C_VEL
LIN {X 0,Y 481.638,Z 226.985,A -85,B 0,C 180,E1 -6888.956,E2 -6888.956} C_VEL
LIN {X 0,Y 481.658,Z 226.99,A -85,B 0,C 180,E1 -6891.994,E2 -6891.994} C_VEL
LIN {X 0,Y 481.697,Z 226.98,A -85,B 0,C 180,E1 -6895.318,E2 -6895.318} C_VEL
LIN {X 0,Y 481.653,Z 226.989,A -85,B 0,C 180,E1 -6898.312,E2 -6898.312} C_VEL
LIN {X 0,Y 481.706,Z 226.978,A -85,B 0,C 180,E1 -6901.218,E2 -6901.218} C_VEL
LIN {X 0,Y 481.682,Z 226.987,A -85,B 0,C 180,E1 -6904.041,E2 -6904.041} C_VEL
LIN {X 0,Y 481.705,Z 227.106,A -85,B 0,C 180,E1 -6905.487,E2 -6905.487} C_VEL
LIN {X 0,Y 483.42,Z 236.353,A -85,B 0,C 180,E1 -6907.34,E2 -6907.34} C_VEL
LIN {X 0,Y 483.317,Z 243.602,A -85,B 0,C 180,E1 -6908.682,E2 -6908.682} C_VEL
LIN {X 0,Y 482.636,Z 261.719,A -85,B 0,C 180,E1 -6911.974,E2 -6911.974} C_VEL
LIN {X 0,Y 482.362,Z 270.273,A -85,B 0,C 180,E1 -6913.474,E2 -6913.474} C_VEL
LIN {X 0,Y 483.787,Z 279.154,A -85,B 0,C 180,E1 -6913.691,E2 -6913.691} C_VEL
LIN {X 0,Y 484.88,Z 286.236,A -85,B 0,C 180,E1 -6913.836,E2 -6913.836} C_VEL
LIN {X 0,Y 484.274,Z 378.319,A -85,B 0,C 180,E1 -6915.233,E2 -6915.233} C_VEL
LIN {X 0,Y 483.95,Z 391.466,A -85,B 0,C 180,E1 -6915.599,E2 -6915.599} C_VEL
LIN {X 0,Y 483.55,Z 404.132,A -85,B 0,C 180,E1 -6916.124,E2 -6916.124} C_VEL
LIN {X 0,Y 483.177,Z 415.708,A -85,B 0,C 180,E1 -6916.777,E2 -6916.777} C_VEL
LIN {X 0,Y 482.737,Z 427.034,A -85,B 0,C 180,E1 -6917.599,E2 -6917.599} C_VEL
LIN {X 0,Y 482.284,Z 437.508,A -85,B 0,C 180,E1 -6918.547,E2 -6918.547} C_VEL
LIN {X 0,Y 481.865,Z 446.067,A -85,B 0,C 180,E1 -6919.495,E2 -6919.495} C_VEL
LIN {X 0,Y 481.534,Z 453.962,A -85,B 0,C 180,E1 -6920.549,E2 -6920.549} C_VEL
LIN {X 0,Y 481.259,Z 461.671,A -85,B 0,C 180,E1 -6921.814,E2 -6921.814} C_VEL
LIN {X 0,Y 481.019,Z 468.768,A -85,B 0,C 180,E1 -6923.287,E2 -6923.287} C_VEL
LIN {X 0,Y 480.963,Z 473.49,A -85,B 0,C 180,E1 -6924.549,E2 -6924.549} C_VEL
LIN {X 0,Y 480.83,Z 477.096,A -85,B 0,C 180,E1 -6925.808,E2 -6925.808} C_VEL
LIN {X 0,Y 480.873,Z 478.958,A -85,B 0,C 180,E1 -6926.648,E2 -6926.648} C_VEL
LIN {X 0,Y 480.791,Z 481.346,A -85,B 0,C 180,E1 -6928.324,E2 -6928.324} C_VEL
LIN {X 0,Y 480.745,Z 482.169,A -85,B 0,C 180,E1 -6929.999,E2 -6929.999} C_VEL
LIN {X 0,Y 480.761,Z 481.953,A -85,B 0,C 180,E1 -6930.837,E2 -6930.837} C_VEL
LIN {X 0,Y 480.791,Z 481.347,A -85,B 0,C 180,E1 -6931.675,E2 -6931.675} C_VEL
LIN {X 0,Y 480.872,Z 478.959,A -85,B 0,C 180,E1 -6933.351,E2 -6933.351} C_VEL
LIN {X 0,Y 480.841,Z 476.026,A -85,B 0,C 180,E1 -6934.61,E2 -6934.61} C_VEL
LIN {X 0,Y 480.962,Z 472.056,A -85,B 0,C 180,E1 -6935.87,E2 -6935.87} C_VEL
LIN {X 0,Y 481.111,Z 465.949,A -85,B 0,C 180,E1 -6937.343,E2 -6937.343} C_VEL
LIN {X 0,Y 481.358,Z 459.275,A -85,B 0,C 180,E1 -6938.606,E2 -6938.606} C_VEL
LIN {X 0,Y 481.692,Z 450.992,A -85,B 0,C 180,E1 -6939.87,E2 -6939.87} C_VEL
LIN {X 0,Y 482.021,Z 442.495,A -85,B 0,C 180,E1 -6940.925,E2 -6940.925} C_VEL
LIN {X 0,Y 482.565,Z 431.997,A -85,B 0,C 180,E1 -6941.977,E2 -6941.977} C_VEL
LIN {X 0,Y 482.888,Z 420.651,A -85,B 0,C 180,E1 -6942.894,E2 -6942.894} C_VEL
LIN {X 0,Y 483.329,Z 410.204,A -85,B 0,C 180,E1 -6943.56,E2 -6943.56} C_VEL
LIN {X 0,Y 483.727,Z 398.467,A -85,B 0,C 180,E1 -6944.138,E2 -6944.138} C_VEL
LIN {X 0,Y 484.1,Z 385.855,A -85,B 0,C 180,E1 -6944.583,E2 -6944.583} C_VEL
LIN {X 0,Y 484.307,Z 372.989,A -85,B 0,C 180,E1 -6944.872,E2 -6944.872} C_VEL
LIN {X 0,Y 484.845,Z 285.331,A -85,B 0,C 180,E1 -6946.192,E2 -6946.192} C_VEL
LIN {X 0,Y 482.401,Z 270.257,A -85,B 0,C 180,E1 -6946.538,E2 -6946.538} C_VEL
LIN {X 0,Y 482.398,Z 266.46,A -85,B 0,C 180,E1 -6947.158,E2 -6947.158} C_VEL
LIN {X 0,Y 482.967,Z 250.578,A -85,B 0,C 180,E1 -6949.996,E2 -6949.996} C_VEL
LIN {X 0,Y 483.489,Z 237.128,A -85,B 0,C 180,E1 -6952.43,E2 -6952.43} C_VEL
LIN {X 0,Y 481.744,Z 227.36,A -85,B 0,C 180,E1 -6954.338,E2 -6954.338} C_VEL
LIN {X 0,Y 481.676,Z 226.989,A -85,B 0,C 180,E1 -6954.571,E2 -6954.571} C_VEL
LIN {X 0,Y 481.696,Z 226.985,A -85,B 0,C 180,E1 -6957.831,E2 -6957.831} C_VEL
LIN {X 0,Y 481.648,Z 226.987,A -85,B 0,C 180,E1 -6960.71,E2 -6960.71} C_VEL
LIN {X 0,Y 481.702,Z 226.983,A -85,B 0,C 180,E1 -6963.732,E2 -6963.732} C_VEL
LIN {X 0,Y 481.623,Z 226.986,A -85,B 0,C 180,E1 -6966.746,E2 -6966.746} C_VEL
LIN {X 0,Y 481.659,Z 226.985,A -85,B 0,C 180,E1 -6969.941,E2 -6969.941} C_VEL
LIN {X 0,Y 481.628,Z 226.986,A -85,B 0,C 180,E1 -6973.144,E2 -6973.144} C_VEL
LIN {X 0,Y 481.655,Z 226.984,A -85,B 0,C 180,E1 -6975.64,E2 -6975.64} C_VEL
LIN {X 0,Y 481.635,Z 226.988,A -85,B 0,C 180,E1 -6978.954,E2 -6978.954} C_VEL
LIN {X 0,Y 481.649,Z 226.984,A -85,B 0,C 180,E1 -6981.992,E2 -6981.992} C_VEL
LIN {X 0,Y 481.681,Z 226.979,A -85,B 0,C 180,E1 -6985.315,E2 -6985.315} C_VEL
LIN {X 0,Y 481.642,Z 226.988,A -85,B 0,C 180,E1 -6988.309,E2 -6988.309} C_VEL
LIN {X 0,Y 481.658,Z 226.984,A -85,B 0,C 180,E1 -6991.214,E2 -6991.214} C_VEL
LIN {X 0,Y 481.641,Z 226.984,A -85,B 0,C 180,E1 -6994.037,E2 -6994.037} C_VEL
LIN {X 0,Y 481.651,Z 226.988,A -85,B 0,C 180,E1 -6996.816,E2 -6996.816} C_VEL
LIN {X 0,Y 481.69,Z 226.981,A -85,B 0,C 180,E1 -6999.5,E2 -6999.5} C_VEL
LIN {X 0,Y 481.683,Z 226.976,A -85,B 0,C 180,E1 -7002.155,E2 -7002.155} C_VEL
LIN {X 0,Y 481.733,Z 226.978,A -85,B 0,C 180,E1 -7004.773,E2 -7004.773} C_VEL
LIN {X 0,Y 481.744,Z 226.971,A -85,B 0,C 180,E1 -7008.212,E2 -7008.212} C_VEL
LIN {X 0,Y 481.712,Z 226.978,A -85,B 0,C 180,E1 -7011.608,E2 -7011.608} C_VEL
LIN {X 0,Y 481.785,Z 226.968,A -85,B 0,C 180,E1 -7014.137,E2 -7014.137} C_VEL
LIN {X 0,Y 481.894,Z 226.958,A -85,B 0,C 180,E1 -7017.49,E2 -7017.49} C_VEL
LIN {X 0,Y 481.895,Z 226.953,A -85,B 0,C 180,E1 -7019.997,E2 -7019.997} C_VEL
LIN {X 0,Y 481.891,Z 226.953,A -85,B 0,C 180,E1 -7022.505,E2 -7022.505} C_VEL
LIN {X 0,Y 481.75,Z 226.976,A -85,B 0,C 180,E1 -7025.858,E2 -7025.858} C_VEL
LIN {X 0,Y 481.701,Z 226.978,A -85,B 0,C 180,E1 -7028.386,E2 -7028.386} C_VEL
LIN {X 0,Y 481.72,Z 226.982,A -85,B 0,C 180,E1 -7031.782,E2 -7031.782} C_VEL
LIN {X 0,Y 481.722,Z 226.976,A -85,B 0,C 180,E1 -7035.221,E2 -7035.221} C_VEL
LIN {X 0,Y 481.687,Z 226.981,A -85,B 0,C 180,E1 -7038.719,E2 -7038.719} C_VEL
LIN {X 0,Y 481.626,Z 226.988,A -85,B 0,C 180,E1 -7041.392,E2 -7041.392} C_VEL
LIN {X 0,Y 481.636,Z 226.992,A -85,B 0,C 180,E1 -7044.111,E2 -7044.111} C_VEL
LIN {X 0,Y 481.673,Z 226.982,A -85,B 0,C 180,E1 -7047.124,E2 -7047.124} C_VEL
LIN {X 0,Y 481.649,Z 226.984,A -85,B 0,C 180,E1 -7049.739,E2 -7049.739} C_VEL
LIN {X 0,Y 481.647,Z 226.989,A -85,B 0,C 180,E1 -7052.671,E2 -7052.671} C_VEL
LIN {X 0,Y 481.616,Z 226.989,A -85,B 0,C 180,E1 -7055.706,E2 -7055.706} C_VEL
LIN {X 0,Y 481.686,Z 226.983,A -85,B 0,C 180,E1 -7059.351,E2 -7059.351} C_VEL
LIN {X 0,Y 481.645,Z 226.99,A -85,B 0,C 180,E1 -7062.155,E2 -7062.155} C_VEL
LIN {X 0,Y 481.689,Z 227.144,A -85,B 0,C 180,E1 -7064.742,E2 -7064.742} C_VEL
LIN {X 0,Y 482.892,Z 233.725,A -85,B 0,C 180,E1 -7066.083,E2 -7066.083} C_VEL
LIN {X 0,Y 482.64,Z 246.658,A -85,B 0,C 180,E1 -7068.507,E2 -7068.507} C_VEL
LIN {X 0,Y 482.375,Z 257.776,A -85,B 0,C 180,E1 -7070.518,E2 -7070.518} C_VEL
LIN {X 0,Y 484.907,Z 272.056,A -85,B 0,C 180,E1 -7070.848,E2 -7070.848} C_VEL
LIN {X 0,Y 484.238,Z 365.704,A -85,B 0,C 180,E1 -7072.279,E2 -7072.279} C_VEL
LIN {X 0,Y 483.988,Z 378.732,A -85,B 0,C 180,E1 -7072.648,E2 -7072.648} C_VEL
LIN {X 0,Y 483.978,Z 379.543,A -85,B 0,C 180,E1 -7072.677,E2 -7072.677} C_VEL
LIN {X 0,Y 483.116,Z 385.182,A -85,B 0,C 180,E1 -7072.868,E2 -7072.868} C_VEL
LIN {X 0,Y 480.059,Z 394.202,A -85,B 0,C 180,E1 -7073.205,E2 -7073.205} C_VEL
LIN {X 0,Y 476.994,Z 402.882,A -85,B 0,C 180,E1 -7073.64,E2 -7073.64} C_VEL
LIN {X 0,Y 476.121,Z 407.981,A -85,B 0,C 180,E1 -7073.98,E2 -7073.98} C_VEL
LIN {X 0,Y 475.596,Z 419.605,A -85,B 0,C 180,E1 -7074.939,E2 -7074.939} C_VEL
LIN {X 0,Y 475.201,Z 429.048,A -85,B 0,C 180,E1 -7075.908,E2 -7075.908} C_VEL
LIN {X 0,Y 474.771,Z 437.833,A -85,B 0,C 180,E1 -7077.008,E2 -7077.008} C_VEL
LIN {X 0,Y 474.394,Z 445.986,A -85,B 0,C 180,E1 -7078.271,E2 -7078.271} C_VEL
LIN {X 0,Y 474.139,Z 453.533,A -85,B 0,C 180,E1 -7079.738,E2 -7079.738} C_VEL
LIN {X 0,Y 473.884,Z 459.796,A -85,B 0,C 180,E1 -7081.349,E2 -7081.349} C_VEL
LIN {X 0,Y 473.771,Z 464.119,A -85,B 0,C 180,E1 -7082.869,E2 -7082.869} C_VEL
LIN {X 0,Y 473.701,Z 465.631,A -85,B 0,C 180,E1 -7083.572,E2 -7083.572} C_VEL
LIN {X 0,Y 473.628,Z 467.601,A -85,B 0,C 180,E1 -7084.833,E2 -7084.833} C_VEL
LIN {X 0,Y 473.553,Z 468.831,A -85,B 0,C 180,E1 -7086.379,E2 -7086.379} C_VEL
LIN {X 0,Y 473.581,Z 468.906,A -85,B 0,C 180,E1 -7087.305,E2 -7087.305} C_VEL
LIN {X 0,Y 473.578,Z 468.546,A -85,B 0,C 180,E1 -7088.223,E2 -7088.223} C_VEL
LIN {X 0,Y 473.623,Z 467.671,A -85,B 0,C 180,E1 -7089.19,E2 -7089.19} C_VEL
LIN {X 0,Y 473.675,Z 466.431,A -85,B 0,C 180,E1 -7090.048,E2 -7090.048} C_VEL
LIN {X 0,Y 473.794,Z 462.964,A -85,B 0,C 180,E1 -7091.669,E2 -7091.669} C_VEL
LIN {X 0,Y 473.926,Z 458.187,A -85,B 0,C 180,E1 -7093.193,E2 -7093.193} C_VEL
LIN {X 0,Y 474.2,Z 451.601,A -85,B 0,C 180,E1 -7094.749,E2 -7094.749} C_VEL
LIN {X 0,Y 474.475,Z 444.424,A -85,B 0,C 180,E1 -7096.073,E2 -7096.073} C_VEL
LIN {X 0,Y 474.845,Z 435.968,A -85,B 0,C 180,E1 -7097.318,E2 -7097.318} C_VEL
LIN {X 0,Y 475.289,Z 426.165,A -85,B 0,C 180,E1 -7098.486,E2 -7098.486} C_VEL
LIN {X 0,Y 475.751,Z 415.929,A -85,B 0,C 180,E1 -7099.467,E2 -7099.467} C_VEL
LIN {X 0,Y 476.251,Z 404.504,A -85,B 0,C 180,E1 -7100.337,E2 -7100.337} C_VEL
LIN {X 0,Y 476.743,Z 391.924,A -85,B 0,C 180,E1 -7101.081,E2 -7101.081} C_VEL
LIN {X 0,Y 477.075,Z 379.008,A -85,B 0,C 180,E1 -7101.636,E2 -7101.636} C_VEL
LIN {X 0,Y 477.356,Z 365.906,A -85,B 0,C 180,E1 -7102.014,E2 -7102.014} C_VEL
LIN {X 0,Y 478.041,Z 281.07,A -85,B 0,C 180,E1 -7103.326,E2 -7103.326} C_VEL
LIN {X 0,Y 477.865,Z 271.33,A -85,B 0,C 180,E1 -7103.482,E2 -7103.482} C_VEL
LIN {X 0,Y 475.473,Z 258.175,A -85,B 0,C 180,E1 -7103.796,E2 -7103.796} C_VEL
LIN {X 0,Y 475.521,Z 255.354,A -85,B 0,C 180,E1 -7104.275,E2 -7104.275} C_VEL
LIN {X 0,Y 476.193,Z 238.324,A -85,B 0,C 180,E1 -7107.675,E2 -7107.675} C_VEL
LIN {X 0,Y 475.994,Z 235.246,A -85,B 0,C 180,E1 -7108.309,E2 -7108.309} C_VEL
LIN {X 0,Y 474.869,Z 227.895,A -85,B 0,C 180,E1 -7109.921,E2 -7109.921} C_VEL
LIN {X 0,Y 474.856,Z 227.835,A -85,B 0,C 180,E1 -7112.545,E2 -7112.545} C_VEL
LIN {X 0,Y 474.743,Z 227.847,A -85,B 0,C 180,E1 -7115.949,E2 -7115.949} C_VEL
LIN {X 0,Y 474.69,Z 227.852,A -85,B 0,C 180,E1 -7118.515,E2 -7118.515} C_VEL
LIN {X 0,Y 474.702,Z 227.85,A -85,B 0,C 180,E1 -7121.963,E2 -7121.963} C_VEL
LIN {X 0,Y 474.644,Z 227.863,A -85,B 0,C 180,E1 -7125.769,E2 -7125.769} C_VEL
LIN {X 0,Y 474.63,Z 227.858,A -85,B 0,C 180,E1 -7129.012,E2 -7129.012} C_VEL
LIN {X 0,Y 474.553,Z 227.872,A -85,B 0,C 180,E1 -7131.731,E2 -7131.731} C_VEL
LIN {X 0,Y 474.603,Z 227.863,A -85,B 0,C 180,E1 -7134.496,E2 -7134.496} C_VEL
LIN {X 0,Y 474.605,Z 227.862,A -85,B 0,C 180,E1 -7137.326,E2 -7137.326} C_VEL
LIN {X 0,Y 474.572,Z 227.868,A -85,B 0,C 180,E1 -7140.233,E2 -7140.233} C_VEL
LIN {X 0,Y 474.585,Z 227.863,A -85,B 0,C 180,E1 -7143.225,E2 -7143.225} C_VEL
LIN {X 0,Y 474.55,Z 227.868,A -85,B 0,C 180,E1 -7146.327,E2 -7146.327} C_VEL
LIN {X 0,Y 474.573,Z 227.865,A -85,B 0,C 180,E1 -7149.647,E2 -7149.647} C_VEL
LIN {X 0,Y 474.549,Z 227.868,A -85,B 0,C 180,E1 -7152.942,E2 -7152.942} C_VEL
LIN {X 0,Y 474.578,Z 227.864,A -85,B 0,C 180,E1 -7155.897,E2 -7155.897} C_VEL
LIN {X 0,Y 474.569,Z 227.862,A -85,B 0,C 180,E1 -7159.343,E2 -7159.343} C_VEL
LIN {X 0,Y 474.588,Z 227.854,A -85,B 0,C 180,E1 -7161.708,E2 -7161.708} C_VEL
LIN {X 0,Y 474.604,Z 227.863,A -85,B 0,C 180,E1 -7164.729,E2 -7164.729} C_VEL
LIN {X 0,Y 474.609,Z 227.859,A -85,B 0,C 180,E1 -7167.79,E2 -7167.79} C_VEL
LIN {X 0,Y 474.58,Z 227.858,A -85,B 0,C 180,E1 -7170.895,E2 -7170.895} C_VEL
LIN {X 0,Y 474.568,Z 227.867,A -85,B 0,C 180,E1 -7173.627,E2 -7173.627} C_VEL
LIN {X 0,Y 474.624,Z 227.859,A -85,B 0,C 180,E1 -7176.646,E2 -7176.646} C_VEL
LIN {X 0,Y 474.643,Z 227.85,A -85,B 0,C 180,E1 -7180.093,E2 -7180.093} C_VEL
LIN {X 0,Y 474.62,Z 227.843,A -85,B 0,C 180,E1 -7182.777,E2 -7182.777} C_VEL
LIN {X 0,Y 474.635,Z 227.855,A -85,B 0,C 180,E1 -7185.424,E2 -7185.424} C_VEL
LIN {X 0,Y 474.689,Z 227.856,A -85,B 0,C 180,E1 -7188.041,E2 -7188.041} C_VEL
LIN {X 0,Y 474.692,Z 227.849,A -85,B 0,C 180,E1 -7191.489,E2 -7191.489} C_VEL
LIN {X 0,Y 474.737,Z 227.836,A -85,B 0,C 180,E1 -7194.055,E2 -7194.055} C_VEL
LIN {X 0,Y 474.872,Z 227.824,A -85,B 0,C 180,E1 -7197.458,E2 -7197.458} C_VEL
LIN {X 0,Y 474.88,Z 227.832,A -85,B 0,C 180,E1 -7200.003,E2 -7200.003} C_VEL
LIN {X 0,Y 474.873,Z 227.825,A -85,B 0,C 180,E1 -7202.548,E2 -7202.548} C_VEL
LIN {X 0,Y 474.752,Z 227.831,A -85,B 0,C 180,E1 -7205.951,E2 -7205.951} C_VEL
LIN {X 0,Y 474.704,Z 227.854,A -85,B 0,C 180,E1 -7208.517,E2 -7208.517} C_VEL
LIN {X 0,Y 474.71,Z 227.849,A -85,B 0,C 180,E1 -7211.965,E2 -7211.965} C_VEL
LIN {X 0,Y 474.687,Z 227.84,A -85,B 0,C 180,E1 -7215.769,E2 -7215.769} C_VEL
LIN {X 0,Y 474.669,Z 227.859,A -85,B 0,C 180,E1 -7219.012,E2 -7219.012} C_VEL
LIN {X 0,Y 474.595,Z 227.86,A -85,B 0,C 180,E1 -7221.731,E2 -7221.731} C_VEL
LIN {X 0,Y 474.636,Z 227.849,A -85,B 0,C 180,E1 -7224.496,E2 -7224.496} C_VEL
LIN {X 0,Y 474.647,Z 227.861,A -85,B 0,C 180,E1 -7227.326,E2 -7227.326} C_VEL
LIN {X 0,Y 474.606,Z 227.858,A -85,B 0,C 180,E1 -7230.232,E2 -7230.232} C_VEL
LIN {X 0,Y 474.624,Z 227.864,A -85,B 0,C 180,E1 -7233.224,E2 -7233.224} C_VEL
LIN {X 0,Y 474.593,Z 227.861,A -85,B 0,C 180,E1 -7236.325,E2 -7236.325} C_VEL
LIN {X 0,Y 474.632,Z 227.866,A -85,B 0,C 180,E1 -7239.549,E2 -7239.549} C_VEL
LIN {X 0,Y 474.598,Z 227.858,A -85,B 0,C 180,E1 -7242.233,E2 -7242.233} C_VEL
LIN {X 0,Y 474.626,Z 227.863,A -85,B 0,C 180,E1 -7245.299,E2 -7245.299} C_VEL
LIN {X 0,Y 474.61,Z 227.863,A -85,B 0,C 180,E1 -7248.213,E2 -7248.213} C_VEL
LIN {X 0,Y 474.618,Z 227.865,A -85,B 0,C 180,E1 -7251.543,E2 -7251.543} C_VEL
LIN {X 0,Y 474.631,Z 227.86,A -85,B 0,C 180,E1 -7254.726,E2 -7254.726} C_VEL
LIN {X 0,Y 474.645,Z 227.861,A -85,B 0,C 180,E1 -7257.788,E2 -7257.788} C_VEL
LIN {X 0,Y 474.631,Z 227.861,A -85,B 0,C 180,E1 -7260.886,E2 -7260.886} C_VEL
LIN {X 0,Y 474.636,Z 227.86,A -85,B 0,C 180,E1 -7263.626,E2 -7263.626} C_VEL
LIN {X 0,Y 474.666,Z 227.957,A -85,B 0,C 180,E1 -7265.274,E2 -7265.274} C_VEL
LIN {X 0,Y 476.442,Z 237.455,A -85,B 0,C 180,E1 -7267.218,E2 -7267.218} C_VEL
LIN {X 0,Y 476.443,Z 243.498,A -85,B 0,C 180,E1 -7268.359,E2 -7268.359} C_VEL
LIN {X 0,Y 475.705,Z 261.613,A -85,B 0,C 180,E1 -7271.702,E2 -7271.702} C_VEL
LIN {X 0,Y 475.371,Z 270.174,A -85,B 0,C 180,E1 -7273.225,E2 -7273.225} C_VEL
LIN {X 0,Y 476.488,Z 277.128,A -85,B 0,C 180,E1 -7273.407,E2 -7273.407} C_VEL
LIN {X 0,Y 478.039,Z 287.947,A -85,B 0,C 180,E1 -7273.628,E2 -7273.628} C_VEL
LIN {X 0,Y 477.405,Z 378.089,A -85,B 0,C 180,E1 -7275.016,E2 -7275.016} C_VEL
LIN {X 0,Y 477.089,Z 391.284,A -85,B 0,C 180,E1 -7275.388,E2 -7275.388} C_VEL
LIN {X 0,Y 476.662,Z 403.975,A -85,B 0,C 180,E1 -7275.919,E2 -7275.919} C_VEL
LIN {X 0,Y 476.245,Z 415.255,A -85,B 0,C 180,E1 -7276.56,E2 -7276.56} C_VEL
LIN {X 0,Y 475.777,Z 426.996,A -85,B 0,C 180,E1 -7277.422,E2 -7277.422} C_VEL
LIN {X 0,Y 475.297,Z 437.384,A -85,B 0,C 180,E1 -7278.377,E2 -7278.377} C_VEL
LIN {X 0,Y 474.869,Z 445.948,A -85,B 0,C 180,E1 -7279.338,E2 -7279.338} C_VEL
LIN {X 0,Y 474.498,Z 453.847,A -85,B 0,C 180,E1 -7280.408,E2 -7280.408} C_VEL
LIN {X 0,Y 474.193,Z 461.561,A -85,B 0,C 180,E1 -7281.691,E2 -7281.691} C_VEL
LIN {X 0,Y 473.935,Z 468.66,A -85,B 0,C 180,E1 -7283.186,E2 -7283.186} C_VEL
LIN {X 0,Y 473.877,Z 473.385,A -85,B 0,C 180,E1 -7284.467,E2 -7284.467} C_VEL
LIN {X 0,Y 473.737,Z 476.993,A -85,B 0,C 180,E1 -7285.745,E2 -7285.745} C_VEL
LIN {X 0,Y 473.767,Z 478.856,A -85,B 0,C 180,E1 -7286.598,E2 -7286.598} C_VEL
LIN {X 0,Y 473.725,Z 480.252,A -85,B 0,C 180,E1 -7287.448,E2 -7287.448} C_VEL
LIN {X 0,Y 473.69,Z 481.854,A -85,B 0,C 180,E1 -7289.149,E2 -7289.149} C_VEL
LIN {X 0,Y 473.671,Z 482.071,A -85,B 0,C 180,E1 -7289.999,E2 -7289.999} C_VEL
LIN {X 0,Y 473.69,Z 481.856,A -85,B 0,C 180,E1 -7290.849,E2 -7290.849} C_VEL
LIN {X 0,Y 473.724,Z 480.255,A -85,B 0,C 180,E1 -7292.55,E2 -7292.55} C_VEL
LIN {X 0,Y 473.767,Z 478.861,A -85,B 0,C 180,E1 -7293.401,E2 -7293.401} C_VEL
LIN {X 0,Y 473.765,Z 475.927,A -85,B 0,C 180,E1 -7294.679,E2 -7294.679} C_VEL
LIN {X 0,Y 473.866,Z 471.957,A -85,B 0,C 180,E1 -7295.958,E2 -7295.958} C_VEL
LIN {X 0,Y 474.033,Z 465.849,A -85,B 0,C 180,E1 -7297.453,E2 -7297.453} C_VEL
